# B&R Automation Studio project NAINV104C00R8L515F00 (part 9)

#### Act_Main_P0201.st
```iecst
(** 2018-12-21 **)
ACTION Act_Main_P0201:
	//LF width 2
	IF p_tyNtParamCurr.bLFProdWidth2Prep THEN
		fUIInRtStatOff(ADR(tyP0201OpsConv.tyOps.tyNumProdWidth2.uiRtStat));
		fUIInRtStatHide(ADR(tyP0201OpsConv.tyOps.tyNumProdWidth.uiRtStat));
	ELSE
		fUIInRtStatHide(ADR(tyP0201OpsConv.tyOps.tyNumProdWidth2.uiRtStat));
		fUIInRtStatOff(ADR(tyP0201OpsConv.tyOps.tyNumProdWidth.uiRtStat));
	END_IF

	IF p_tyNtParamCurr.tyDOSettings.diTLGreen<>0 OR p_tyNtParamCurr.tyDOSettings.diTLAmber<>0 OR p_tyNtParamCurr.tyDOSettings.diTLRed<>0 THEN
		IF p_tyNtParamCurr.eTLBuzMode=TLBuzModBHTC THEN
			tyP0201OpsConv.tyOps.tyBitmapMc.usiValueIdx := 200;
		ELSE
			tyP0201OpsConv.tyOps.tyBitmapMc.usiValueIdx := 100;
		END_IF
	ELSE
		tyP0201OpsConv.tyOps.tyBitmapMc.usiValueIdx := 0;
	END_IF

	fUIInRtStatHide(ADR(tyP0200OpsGen.tyOps.tyTxtLdrInActiveCtrl.uiRtStat));
	fUIInRtStatHide(ADR(tyP0201OpsConv.tyOps.tyTxtLdrInActiveCtrl.uiRtStat));
	fUIInRtStatHide(ADR(tyP0200OpsGen.tyOps.tyBitmapWarningLF.uiRtStat));
	fUIInRtStatHide(ADR(tyP0201OpsConv.tyOps.tyBitmapWarningLF.uiRtStat));

	//IO Monitor Standard
	//Digital Input Used
	IF p_tyNtParamCurr.tyDISettings.diSafetyRlySig = 0 THEN
		fUIInRtStatHide(ADR(tyP0201OpsConv.tyIOMonitor.tyBtnSafetyRlySig.uiRtStat));
	END_IF

	IF p_tyNtParamCurr.tyDISettings.diEStopSig = 0 THEN
		fUIInRtStatHide(ADR(tyP0201OpsConv.tyIOMonitor.tyBtnEStop.uiRtStat));
	END_IF

	IF p_tyNtParamCurr.tyDISettings.diCoverSWSig = 0 THEN
		fUIInRtStatHide(ADR(tyP0201OpsConv.tyIOMonitor.tyBtnCoverSWSig.uiRtStat));
	END_IF

	IF p_tyNtParamCurr.tyDISettings.diUBA = 0 THEN
		fUIInRtStatHide(ADR(tyP0201OpsConv.tyIOMonitor.tyBtnUBA.uiRtStat));
	END_IF

	IF p_tyNtParamCurr.tyDISettings.diDSB = 0 THEN
		fUIInRtStatHide(ADR(tyP0201OpsConv.tyIOMonitor.tyBtnDSB.uiRtStat));
	END_IF

	IF p_tyNtParamCurr.tyDISettings.diUBAStat = FALSE THEN
		fUIInRtStatHide(ADR(tyP0201OpsConv.tyIOMonitor.tyBtnUBAStat.uiRtStat));
	END_IF

	IF p_tyNtParamCurr.tyDISettings.diConvLftSen = 0 THEN
		fUIInRtStatHide(ADR(tyP0201OpsConv.tyIOMonitor.tyBtnConvLftSen.uiRtStat));
	END_IF

	IF p_tyNtParamCurr.tyDISettings.diConvRgtSen = 0 THEN
		fUIInRtStatHide(ADR(tyP0201OpsConv.tyIOMonitor.tyBtnConvRgtSen.uiRtStat));
	END_IF

	IF p_tyNtParamCurr.tyDISettings.diPressureSW = 0 THEN
		fUIInRtStatHide(ADR(tyP0201OpsConv.tyIOMonitor.tyBtnPressureSW.uiRtStat));
	END_IF

	IF p_tyNtParamCurr.tyDISettings.diThermalPrtSig = 0 THEN
		fUIInRtStatHide(ADR(tyP0201OpsConv.tyIOMonitor.tyBtnThermalPrtSig.uiRtStat));
	END_IF

	IF p_tyNtParamCurr.tyDISettings.diCoatingSen = 0 THEN
		fUIInRtStatHide(ADR(tyP0201OpsConv.tyIOMonitor.tyBtnCoatingSen.uiRtStat));
	END_IF

	IF p_tyNtParamCurr.tyDISettings.diUSWidthChkSen = 0 THEN
		fUIInRtStatHide(ADR(tyP0201OpsConv.tyIOMonitor.tyBtnUSWidthChkSen.uiRtStat));
	END_IF

	IF p_tyNtParamCurr.tyDISettings.diDSWidthChkSen = 0 THEN
		fUIInRtStatHide(ADR(tyP0201OpsConv.tyIOMonitor.tyBtnDSWidthChkSen.uiRtStat));
	END_IF

	IF p_tyNtParamCurr.tyDISettings.diInvertHomeSen = 0 THEN
		fUIInRtStatHide(ADR(tyP0201OpsConv.tyIOMonitor.tyBtnInvertHomeSen.uiRtStat));
	END_IF

	IF p_tyNtParamCurr.tyDISettings.diInvertRemoteSen = 0 THEN
		fUIInRtStatHide(ADR(tyP0201OpsConv.tyIOMonitor.tyBtnInvertRemoteSen.uiRtStat));
	END_IF

	IF p_tyNtParamCurr.tyDISettings.diInShutterOpenRS = 0 THEN
		fUIInRtStatHide(ADR(tyP0201OpsConv.tyIOMonitor.tyBtnInletShutterOpenRS.uiRtStat));
	END_IF

	IF p_tyNtParamCurr.tyDISettings.diInShutterCloseRS = 0 THEN
		fUIInRtStatHide(ADR(tyP0201OpsConv.tyIOMonitor.tyBtnInletShutterCloseRS.uiRtStat));
	END_IF

	IF p_tyNtParamCurr.tyDISettings.diOutShutterOpenRS = 0 THEN
		fUIInRtStatHide(ADR(tyP0201OpsConv.tyIOMonitor.tyBtnOutletShutterOpenRS.uiRtStat));
	END_IF

	IF p_tyNtParamCurr.tyDISettings.diOutShutterCloseRS = 0 THEN
		fUIInRtStatHide(ADR(tyP0201OpsConv.tyIOMonitor.tyBtnOutletShutterCloseRS.uiRtStat));
	END_IF

	//Digital Output Selected
	IF p_tyNtParamCurr.tyDOSettings.diSafetyRlyRst = 0 THEN
		fUIInRtStatHide(ADR(tyP0201OpsConv.tyIOMonitor.tyBtnSafetyRlyRst.uiRtStat));
	END_IF

	IF p_tyNtParamCurr.tyDOSettings.diTLGreen = 0 THEN
		fUIInRtStatHide(ADR(tyP0201OpsConv.tyIOMonitor.tyBtnTLGreen.uiRtStat));
	END_IF

	IF p_tyNtParamCurr.tyDOSettings.diTLAmber = 0 THEN
		fUIInRtStatHide(ADR(tyP0201OpsConv.tyIOMonitor.tyBtnTLAmber.uiRtStat));
	END_IF

	IF p_tyNtParamCurr.tyDOSettings.diTLRed = 0 THEN
		fUIInRtStatHide(ADR(tyP0201OpsConv.tyIOMonitor.tyBtnTLRed.uiRtStat));
	END_IF

	IF p_tyNtParamCurr.tyDOSettings.diTLWhite = 0 THEN
		fUIInRtStatHide(ADR(tyP0201OpsConv.tyIOMonitor.tyBtnTLWhite.uiRtStat));
	END_IF

	IF p_tyNtParamCurr.tyDOSettings.diTLBlue = 0 THEN
		fUIInRtStatHide(ADR(tyP0201OpsConv.tyIOMonitor.tyBtnTLBlue.uiRtStat));
	END_IF

	IF p_tyNtParamCurr.tyDOSettings.diBuz = 0 THEN
		fUIInRtStatHide(ADR(tyP0201OpsConv.tyIOMonitor.tyBtnBuzzer.uiRtStat));
	END_IF

	IF p_tyNtParamCurr.tyDOSettings.diCoatingStprRet = 0 THEN
		fUIInRtStatHide(ADR(tyP0201OpsConv.tyIOMonitor.tyBtnCoatingRetCtrl.uiRtStat));
	END_IF

	IF p_tyNtParamCurr.tyDOSettings.diUSB = 0 THEN
		fUIInRtStatHide(ADR(tyP0201OpsConv.tyIOMonitor.tyBtnUSB.uiRtStat));
	END_IF

	IF p_tyNtParamCurr.tyDOSettings.diDBA = 0 THEN
		fUIInRtStatHide(ADR(tyP0201OpsConv.tyIOMonitor.tyBtnDBA.uiRtStat));
	END_IF

	IF p_tyNtParamCurr.tyDOSettings.diDBAStat = 0 THEN
		fUIInRtStatHide(ADR(tyP0201OpsConv.tyIOMonitor.tyBtnDBAStat.uiRtStat));
	END_IF

	IF p_tyNtParamCurr.tyDOSettings.diConvMtrCW = 0 THEN
		fUIInRtStatHide(ADR(tyP0201OpsConv.tyIOMonitor.tyBtnConvMtrCW.uiRtStat));
	END_IF

	IF p_tyNtParamCurr.tyDOSettings.diConvMtrCCW = 0 THEN
		fUIInRtStatHide(ADR(tyP0201OpsConv.tyIOMonitor.tyBtnConvMtrCCW.uiRtStat));
	END_IF

	IF p_tyNtParamCurr.tyDOSettings.diStprUnblkCtrl = 0 THEN
		fUIInRtStatHide(ADR(tyP0201OpsConv.tyIOMonitor.tyBtnStprUnblkCtrl.uiRtStat));
	END_IF

	IF p_tyNtParamCurr.tyDOSettings.diStprBlkCtrl = 0 THEN
		fUIInRtStatHide(ADR(tyP0201OpsConv.tyIOMonitor.tyBtnStprBlkCtrl.uiRtStat));
	END_IF

	IF p_tyNtParamCurr.tyDOSettings.diInvertBrake = 0 THEN
		fUIInRtStatHide(ADR(tyP0201OpsConv.tyIOMonitor.tyBtnInvertBrake.uiRtStat));
	END_IF

	IF p_tyNtParamCurr.tyDOSettings.diInvertHome = 0 THEN
		fUIInRtStatHide(ADR(tyP0201OpsConv.tyIOMonitor.tyBtnInvertHome.uiRtStat));
	END_IF

	IF p_tyNtParamCurr.tyDOSettings.diInvertRemote = 0 THEN
		fUIInRtStatHide(ADR(tyP0201OpsConv.tyIOMonitor.tyBtnInvertRemote.uiRtStat));
	END_IF

	IF p_tyNtParamCurr.tyDOSettings.diMtrPwrRly = 0 THEN
		fUIInRtStatHide(ADR(tyP0201OpsConv.tyIOMonitor.tyBtnMtrPwrRly.uiRtStat));
	END_IF

	IF p_tyNtParamCurr.tyDOSettings.diClampControl = 0 THEN
		fUIInRtStatHide(ADR(tyP0201OpsConv.tyIOMonitor.tyBtnClampCtrl.uiRtStat));
	END_IF

	IF p_tyNtParamCurr.tyDOSettings.diUnclampControl = 0 THEN
		fUIInRtStatHide(ADR(tyP0201OpsConv.tyIOMonitor.tyBtnUnclampCtrl.uiRtStat));
	END_IF

	IF p_tyNtParamCurr.tyDOSettings.diInShutterOpenCtrl = 0 THEN
		fUIInRtStatHide(ADR(tyP0201OpsConv.tyIOMonitor.tyBtnInShutterOpenCtrl.uiRtStat));
	END_IF

	IF p_tyNtParamCurr.tyDOSettings.diInShutterCloseCtrl = 0 THEN
		fUIInRtStatHide(ADR(tyP0201OpsConv.tyIOMonitor.tyBtnInShutterCloseCtrl.uiRtStat));
	END_IF

	IF p_tyNtParamCurr.tyDOSettings.diOutShutterOpenCtrl = 0 THEN
		fUIInRtStatHide(ADR(tyP0201OpsConv.tyIOMonitor.tyBtnOutShutterOpenCtrl.uiRtStat));
	END_IF

	IF p_tyNtParamCurr.tyDOSettings.diOutShutterCloseCtrl = 0 THEN
		fUIInRtStatHide(ADR(tyP0201OpsConv.tyIOMonitor.tyBtnOutShutterCloseCtrl.uiRtStat));
	END_IF

	//IO Monitor Non Standard
	//Digital Input Used
	IF p_tyNtParamCurr.tyDISettings.diSafetyRlySig = 0 THEN
		fUIInRtStatHide(ADR(tyP0201OpsConv.tyIOMonitorXStd.tyBtnSafetyRlySig.uiRtStat));
	END_IF

	IF p_tyNtParamCurr.tyDISettings.diEStopSig = 0 THEN
		fUIInRtStatHide(ADR(tyP0201OpsConv.tyIOMonitorXStd.tyBtnEStop.uiRtStat));
	END_IF

	IF p_tyNtParamCurr.tyDISettings.diCoverSWSig = 0 THEN
		fUIInRtStatHide(ADR(tyP0201OpsConv.tyIOMonitorXStd.tyBtnCoverSWSig.uiRtStat));
	END_IF

	IF p_tyNtParamCurr.tyDISettings.diUBA = 0 THEN
		fUIInRtStatHide(ADR(tyP0201OpsConv.tyIOMonitorXStd.tyBtnUBA.uiRtStat));
	END_IF

	IF p_tyNtParamCurr.tyDISettings.diUBA2 = 0 THEN
		fUIInRtStatHide(ADR(tyP0201OpsConv.tyIOMonitorXStd.tyBtnUBA2.uiRtStat));
	END_IF

	IF p_tyNtParamCurr.tyDISettings.diDSB = 0 THEN
		fUIInRtStatHide(ADR(tyP0201OpsConv.tyIOMonitorXStd.tyBtnDSB.uiRtStat));
	END_IF

	IF p_tyNtParamCurr.tyDISettings.diUBAStat = FALSE THEN
		fUIInRtStatHide(ADR(tyP0201OpsConv.tyIOMonitorXStd.tyBtnUBAStat.uiRtStat));
	END_IF

	IF p_tyNtParamCurr.tyDISettings.diUBAStat2 = FALSE THEN
		fUIInRtStatHide(ADR(tyP0201OpsConv.tyIOMonitorXStd.tyBtnUBAStat2.uiRtStat));
	END_IF

	IF p_tyNtParamCurr.tyDISettings.diConvLftSen = 0 THEN
		fUIInRtStatHide(ADR(tyP0201OpsConv.tyIOMonitorXStd.tyBtnConvLftSen.uiRtStat));
	END_IF

	IF p_tyNtParamCurr.tyDISettings.diConvRgtSen = 0 THEN
		fUIInRtStatHide(ADR(tyP0201OpsConv.tyIOMonitorXStd.tyBtnConvRgtSen.uiRtStat));
	END_IF

	IF p_tyNtParamCurr.tyDISettings.diPressureSW = 0 THEN
		fUIInRtStatHide(ADR(tyP0201OpsConv.tyIOMonitorXStd.tyBtnPressureSW.uiRtStat));
	END_IF

	IF p_tyNtParamCurr.tyDISettings.diThermalPrtSig = 0 THEN
		fUIInRtStatHide(ADR(tyP0201OpsConv.tyIOMonitorXStd.tyBtnThermalPrtSig.uiRtStat));
	END_IF

	IF p_tyNtParamCurr.tyDISettings.diCoatingSen = 0 THEN
		fUIInRtStatHide(ADR(tyP0201OpsConv.tyIOMonitorXStd.tyBtnCoatingSen.uiRtStat));
	END_IF

	IF p_tyNtParamCurr.tyDISettings.diUSWidthChkSen = 0 THEN
		fUIInRtStatHide(ADR(tyP0201OpsConv.tyIOMonitorXStd.tyBtnUSWidthChkSen.uiRtStat));
	END_IF

	IF p_tyNtParamCurr.tyDISettings.diDSWidthChkSen = 0 THEN
		fUIInRtStatHide(ADR(tyP0201OpsConv.tyIOMonitorXStd.tyBtnDSWidthChkSen.uiRtStat));
	END_IF

	IF p_tyNtParamCurr.tyDISettings.diInvertHomeSen = 0 THEN
		fUIInRtStatHide(ADR(tyP0201OpsConv.tyIOMonitorXStd.tyBtnInvertHomeSen.uiRtStat));
	END_IF

	IF p_tyNtParamCurr.tyDISettings.diInvertRemoteSen = 0 THEN
		fUIInRtStatHide(ADR(tyP0201OpsConv.tyIOMonitorXStd.tyBtnInvertRemoteSen.uiRtStat));
	END_IF

	IF p_tyNtParamCurr.tyDISettings.diInShutterOpenRS = 0 THEN
		fUIInRtStatHide(ADR(tyP0201OpsConv.tyIOMonitorXStd.tyBtnInletShutterOpenRS.uiRtStat));
	END_IF

	IF p_tyNtParamCurr.tyDISettings.diInShutterCloseRS = 0 THEN
		fUIInRtStatHide(ADR(tyP0201OpsConv.tyIOMonitorXStd.tyBtnInletShutterCloseRS.uiRtStat));
	END_IF

	IF p_tyNtParamCurr.tyDISettings.diOutShutterOpenRS = 0 THEN
		fUIInRtStatHide(ADR(tyP0201OpsConv.tyIOMonitorXStd.tyBtnOutletShutterOpenRS.uiRtStat));
	END_IF

	IF p_tyNtParamCurr.tyDISettings.diOutShutterCloseRS = 0 THEN
		fUIInRtStatHide(ADR(tyP0201OpsConv.tyIOMonitorXStd.tyBtnOutletShutterCloseRS.uiRtStat));
	END_IF

	IF p_tyNtParamCurr.tyDISettings.diClamp2Sen = 0 THEN
		fUIInRtStatHide(ADR(tyP0201OpsConv.tyIOMonitorXStd.tyBtnClamp2Sen.uiRtStat));
	END_IF

	IF p_tyNtParamCurr.tyDISettings.diClamp3Sen = 0 THEN
		fUIInRtStatHide(ADR(tyP0201OpsConv.tyIOMonitorXStd.tyBtnClamp3Sen.uiRtStat));
	END_IF

	IF p_tyNtParamCurr.tyDISettings.diClampRS1 = 0 THEN
		fUIInRtStatHide(ADR(tyP0201OpsConv.tyIOMonitorXStd.tyBtnClampRS1.uiRtStat));
	END_IF

	IF p_tyNtParamCurr.tyDISettings.diUnClampRS1 = 0 THEN
		fUIInRtStatHide(ADR(tyP0201OpsConv.tyIOMonitorXStd.tyBtnUnClampRS1.uiRtStat));
	END_IF

	IF p_tyNtParamCurr.tyDISettings.diClampRS2 = 0 THEN
		fUIInRtStatHide(ADR(tyP0201OpsConv.tyIOMonitorXStd.tyBtnClampRS2.uiRtStat));
	END_IF

	IF p_tyNtParamCurr.tyDISettings.diUnClampRS2 = 0 THEN
		fUIInRtStatHide(ADR(tyP0201OpsConv.tyIOMonitorXStd.tyBtnUnClampRS2.uiRtStat));
	END_IF

	IF p_tyNtParamCurr.tyDISettings.diClampRS3 = 0 THEN
		fUIInRtStatHide(ADR(tyP0201OpsConv.tyIOMonitorXStd.tyBtnClampRS3.uiRtStat));
	END_IF

	IF p_tyNtParamCurr.tyDISettings.diUnClampRS3 = 0 THEN
		fUIInRtStatHide(ADR(tyP0201OpsConv.tyIOMonitorXStd.tyBtnUnClampRS3.uiRtStat));
	END_IF

	//Digital Output Selected
	IF p_tyNtParamCurr.tyDOSettings.diSafetyRlyRst = 0 THEN
		fUIInRtStatHide(ADR(tyP0201OpsConv.tyIOMonitorXStd.tyBtnSafetyRlyRst.uiRtStat));
	END_IF

	IF p_tyNtParamCurr.tyDOSettings.diTLGreen = 0 THEN
		fUIInRtStatHide(ADR(tyP0201OpsConv.tyIOMonitorXStd.tyBtnTLGreen.uiRtStat));
	END_IF

	IF p_tyNtParamCurr.tyDOSettings.diTLAmber = 0 THEN
		fUIInRtStatHide(ADR(tyP0201OpsConv.tyIOMonitorXStd.tyBtnTLAmber.uiRtStat));
	END_IF

	IF p_tyNtParamCurr.tyDOSettings.diTLRed = 0 THEN
		fUIInRtStatHide(ADR(tyP0201OpsConv.tyIOMonitorXStd.tyBtnTLRed.uiRtStat));
	END_IF

	IF p_tyNtParamCurr.tyDOSettings.diTLWhite = 0 THEN
		fUIInRtStatHide(ADR(tyP0201OpsConv.tyIOMonitorXStd.tyBtnTLWhite.uiRtStat));
	END_IF

	IF p_tyNtParamCurr.tyDOSettings.diTLBlue = 0 THEN
		fUIInRtStatHide(ADR(tyP0201OpsConv.tyIOMonitorXStd.tyBtnTLBlue.uiRtStat));
	END_IF

	IF p_tyNtParamCurr.tyDOSettings.diBuz = 0 THEN
		fUIInRtStatHide(ADR(tyP0201OpsConv.tyIOMonitorXStd.tyBtnBuzzer.uiRtStat));
	END_IF

	IF p_tyNtParamCurr.tyDOSettings.diCoatingStprRet = 0 THEN
		fUIInRtStatHide(ADR(tyP0201OpsConv.tyIOMonitorXStd.tyBtnCoatingRetCtrl.uiRtStat));
	END_IF

	IF p_tyNtParamCurr.tyDOSettings.diUSB = 0 THEN
		fUIInRtStatHide(ADR(tyP0201OpsConv.tyIOMonitorXStd.tyBtnUSB.uiRtStat));
	END_IF

	IF p_tyNtParamCurr.tyDOSettings.diUSB2 = 0 THEN
		fUIInRtStatHide(ADR(tyP0201OpsConv.tyIOMonitorXStd.tyBtnUSB2.uiRtStat));
	END_IF

	IF p_tyNtParamCurr.tyDOSettings.diDBA = 0 THEN
		fUIInRtStatHide(ADR(tyP0201OpsConv.tyIOMonitorXStd.tyBtnDBA.uiRtStat));
	END_IF

	IF p_tyNtParamCurr.tyDOSettings.diDBAStat = 0 THEN
		fUIInRtStatHide(ADR(tyP0201OpsConv.tyIOMonitorXStd.tyBtnDBAStat.uiRtStat));
	END_IF

	IF p_tyNtParamCurr.tyDOSettings.diConvMtrCW = 0 THEN
		fUIInRtStatHide(ADR(tyP0201OpsConv.tyIOMonitorXStd.tyBtnConvMtrCW.uiRtStat));
	END_IF

	IF p_tyNtParamCurr.tyDOSettings.diConvMtrCCW = 0 THEN
		fUIInRtStatHide(ADR(tyP0201OpsConv.tyIOMonitorXStd.tyBtnConvMtrCCW.uiRtStat));
	END_IF

	IF p_tyNtParamCurr.tyDOSettings.diInvertBrake = 0 THEN
		fUIInRtStatHide(ADR(tyP0201OpsConv.tyIOMonitorXStd.tyBtnInvertBrake.uiRtStat));
	END_IF

	IF p_tyNtParamCurr.tyDOSettings.diInvertHome = 0 THEN
		fUIInRtStatHide(ADR(tyP0201OpsConv.tyIOMonitorXStd.tyBtnInvertHome.uiRtStat));
	END_IF

	IF p_tyNtParamCurr.tyDOSettings.diInvertRemote = 0 THEN
		fUIInRtStatHide(ADR(tyP0201OpsConv.tyIOMonitorXStd.tyBtnInvertRemote.uiRtStat));
	END_IF

	IF p_tyNtParamCurr.tyDOSettings.diMtrPwrRly = 0 THEN
		fUIInRtStatHide(ADR(tyP0201OpsConv.tyIOMonitorXStd.tyBtnMtrPwrRly.uiRtStat));
	END_IF

	IF p_tyNtParamCurr.tyDOSettings.diInShutterOpenCtrl = 0 THEN
		fUIInRtStatHide(ADR(tyP0201OpsConv.tyIOMonitorXStd.tyBtnInShutterOpenCtrl.uiRtStat));
	END_IF

	IF p_tyNtParamCurr.tyDOSettings.diInShutterCloseCtrl = 0 THEN
		fUIInRtStatHide(ADR(tyP0201OpsConv.tyIOMonitorXStd.tyBtnInShutterCloseCtrl.uiRtStat));
	END_IF

	IF p_tyNtParamCurr.tyDOSettings.diOutShutterOpenCtrl = 0 THEN
		fUIInRtStatHide(ADR(tyP0201OpsConv.tyIOMonitorXStd.tyBtnOutShutterOpenCtrl.uiRtStat));
	END_IF

	IF p_tyNtParamCurr.tyDOSettings.diOutShutterCloseCtrl = 0 THEN
		fUIInRtStatHide(ADR(tyP0201OpsConv.tyIOMonitorXStd.tyBtnOutShutterCloseCtrl.uiRtStat));
	END_IF

	IF p_tyNtParamCurr.tyDOSettings.diClamp1Ctrl = 0 THEN
		fUIInRtStatHide(ADR(tyP0201OpsConv.tyIOMonitorXStd.tyBtnClamp1Ctrl.uiRtStat));
	END_IF

	IF p_tyNtParamCurr.tyDOSettings.diUnClamp1Ctrl = 0 THEN
		fUIInRtStatHide(ADR(tyP0201OpsConv.tyIOMonitorXStd.tyBtnUnclamp1Ctrl.uiRtStat));
	END_IF

	IF p_tyNtParamCurr.tyDOSettings.diClamp2Ctrl = 0 THEN
		fUIInRtStatHide(ADR(tyP0201OpsConv.tyIOMonitorXStd.tyBtnClamp2Ctrl.uiRtStat));
	END_IF

	IF p_tyNtParamCurr.tyDOSettings.diUnClamp2Ctrl = 0 THEN
		fUIInRtStatHide(ADR(tyP0201OpsConv.tyIOMonitorXStd.tyBtnUnclamp2Ctrl.uiRtStat));
	END_IF

	IF p_tyNtParamCurr.tyDOSettings.diClamp3Ctrl = 0 THEN
		fUIInRtStatHide(ADR(tyP0201OpsConv.tyIOMonitorXStd.tyBtnClamp3Ctrl.uiRtStat));
	END_IF

	IF p_tyNtParamCurr.tyDOSettings.diUnClamp3Ctrl = 0 THEN
		fUIInRtStatHide(ADR(tyP0201OpsConv.tyIOMonitorXStd.tyBtnUnclamp3Ctrl.uiRtStat));
	END_IF

	//XStd Machine Safety
	//Digital Input Used
	IF p_tyNtParamCurr.tyDISettings.diSafetyRlySig = 0 THEN
		fUIInRtStatHide(ADR(tyP0201OpsConv.tyIOMonitorXStdMachineSafety.tyBtnSafetyRlySig.uiRtStat));
	END_IF

	IF p_tyNtParamCurr.tyDISettings.diEStopSig = 0 THEN
		fUIInRtStatHide(ADR(tyP0201OpsConv.tyIOMonitorXStdMachineSafety.tyBtnEStop.uiRtStat));
	END_IF

	IF p_tyNtParamCurr.tyDISettings.diCoverSWSig = 0 THEN
		fUIInRtStatHide(ADR(tyP0201OpsConv.tyIOMonitorXStdMachineSafety.tyBtnCoverSWSig.uiRtStat));
	END_IF

	IF p_tyNtParamCurr.tyDISettings.diUBA = 0 THEN
		fUIInRtStatHide(ADR(tyP0201OpsConv.tyIOMonitorXStdMachineSafety.tyBtnUBA.uiRtStat));
	END_IF

	IF p_tyNtParamCurr.tyDISettings.diDSB = 0 THEN
		fUIInRtStatHide(ADR(tyP0201OpsConv.tyIOMonitorXStdMachineSafety.tyBtnDSB.uiRtStat));
	END_IF

	IF p_tyNtParamCurr.tyDISettings.diUBAStat = FALSE THEN
		fUIInRtStatHide(ADR(tyP0201OpsConv.tyIOMonitorXStdMachineSafety.tyBtnUBAStat.uiRtStat));
	END_IF

	IF p_tyNtParamCurr.tyDISettings.diConvLftSen = 0 THEN
		fUIInRtStatHide(ADR(tyP0201OpsConv.tyIOMonitorXStdMachineSafety.tyBtnConvLftSen.uiRtStat));
	END_IF

	IF p_tyNtParamCurr.tyDISettings.diConvRgtSen = 0 THEN
		fUIInRtStatHide(ADR(tyP0201OpsConv.tyIOMonitorXStdMachineSafety.tyBtnConvRgtSen.uiRtStat));
	END_IF

	IF p_tyNtParamCurr.tyDISettings.diPressureSW = 0 THEN
		fUIInRtStatHide(ADR(tyP0201OpsConv.tyIOMonitorXStdMachineSafety.tyBtnPressureSW.uiRtStat));
	END_IF

	IF p_tyNtParamCurr.tyDISettings.diThermalPrtSig = 0 THEN
		fUIInRtStatHide(ADR(tyP0201OpsConv.tyIOMonitorXStdMachineSafety.tyBtnThermalPrtSig.uiRtStat));
	END_IF

	IF p_tyNtParamCurr.tyDISettings.diCoatingSen = 0 THEN
		fUIInRtStatHide(ADR(tyP0201OpsConv.tyIOMonitorXStdMachineSafety.tyBtnCoatingSen.uiRtStat));
	END_IF

	IF p_tyNtParamCurr.tyDISettings.diUSWidthChkSen = 0 THEN
		fUIInRtStatHide(ADR(tyP0201OpsConv.tyIOMonitorXStdMachineSafety.tyBtnUSWidthChkSen.uiRtStat));
	END_IF

	IF p_tyNtParamCurr.tyDISettings.diDSWidthChkSen = 0 THEN
		fUIInRtStatHide(ADR(tyP0201OpsConv.tyIOMonitorXStdMachineSafety.tyBtnDSWidthChkSen.uiRtStat));
	END_IF

	IF p_tyNtParamCurr.tyDISettings.diInvertHomeSen = 0 THEN
		fUIInRtStatHide(ADR(tyP0201OpsConv.tyIOMonitorXStdMachineSafety.tyBtnInvertHomeSen.uiRtStat));
	END_IF

	IF p_tyNtParamCurr.tyDISettings.diInvertRemoteSen = 0 THEN
		fUIInRtStatHide(ADR(tyP0201OpsConv.tyIOMonitorXStdMachineSafety.tyBtnInvertRemoteSen.uiRtStat));
	END_IF

	IF p_tyNtParamCurr.tyDISettings.diInShutterOpenRS = 0 THEN
		fUIInRtStatHide(ADR(tyP0201OpsConv.tyIOMonitorXStdMachineSafety.tyBtnInletShutterOpenRS.uiRtStat));
	END_IF

	IF p_tyNtParamCurr.tyDISettings.diInShutterCloseRS = 0 THEN
		fUIInRtStatHide(ADR(tyP0201OpsConv.tyIOMonitorXStdMachineSafety.tyBtnInletShutterCloseRS.uiRtStat));
	END_IF

	IF p_tyNtParamCurr.tyDISettings.diOutShutterOpenRS = 0 THEN
		fUIInRtStatHide(ADR(tyP0201OpsConv.tyIOMonitorXStdMachineSafety.tyBtnOutletShutterOpenRS.uiRtStat));
	END_IF

	IF p_tyNtParamCurr.tyDISettings.diOutShutterCloseRS = 0 THEN
		fUIInRtStatHide(ADR(tyP0201OpsConv.tyIOMonitorXStdMachineSafety.tyBtnOutletShutterCloseRS.uiRtStat));
	END_IF

	IF p_tyNtParamCurr.tyDISettings.diClamp2Sen = 0 THEN
		fUIInRtStatHide(ADR(tyP0201OpsConv.tyIOMonitorXStdMachineSafety.tyBtnClamp2Sen.uiRtStat));
	END_IF

	IF p_tyNtParamCurr.tyDISettings.diClamp3Sen = 0 THEN
		fUIInRtStatHide(ADR(tyP0201OpsConv.tyIOMonitorXStdMachineSafety.tyBtnClamp3Sen.uiRtStat));
	END_IF

	IF p_tyNtParamCurr.tyDISettings.diClampRS1 = 0 THEN
		fUIInRtStatHide(ADR(tyP0201OpsConv.tyIOMonitorXStdMachineSafety.tyBtnClampRS1.uiRtStat));
	END_IF

	IF p_tyNtParamCurr.tyDISettings.diUnClampRS1 = 0 THEN
		fUIInRtStatHide(ADR(tyP0201OpsConv.tyIOMonitorXStdMachineSafety.tyBtnUnClampRS1.uiRtStat));
	END_IF

	IF p_tyNtParamCurr.tyDISettings.diClampRS2 = 0 THEN
		fUIInRtStatHide(ADR(tyP0201OpsConv.tyIOMonitorXStdMachineSafety.tyBtnClampRS2.uiRtStat));
	END_IF

	IF p_tyNtParamCurr.tyDISettings.diUnClampRS2 = 0 THEN
		fUIInRtStatHide(ADR(tyP0201OpsConv.tyIOMonitorXStdMachineSafety.tyBtnUnClampRS2.uiRtStat));
	END_IF

	IF p_tyNtParamCurr.tyDISettings.diClampRS3 = 0 THEN
		fUIInRtStatHide(ADR(tyP0201OpsConv.tyIOMonitorXStdMachineSafety.tyBtnClampRS3.uiRtStat));
	END_IF

	IF p_tyNtParamCurr.tyDISettings.diUnClampRS3 = 0 THEN
		fUIInRtStatHide(ADR(tyP0201OpsConv.tyIOMonitorXStdMachineSafety.tyBtnUnClampRS3.uiRtStat));
	END_IF
	// ADD
	IF p_tyNtParamCurr.tyDISettings.diCoverSWSig2 = 0 THEN
		fUIInRtStatHide(ADR(tyP0201OpsConv.tyIOMonitorXStdMachineSafety.tyBtnCoverSWSig2.uiRtStat));
	END_IF

	IF p_tyNtParamCurr.tyDISettings.diSafetySigFromUS = 0 THEN
		fUIInRtStatHide(ADR(tyP0201OpsConv.tyIOMonitorXStdMachineSafety.tyBtnSafetySigFromUS.uiRtStat));
	END_IF

	IF p_tyNtParamCurr.tyDISettings.diSafetySigFromDS = 0 THEN
		fUIInRtStatHide(ADR(tyP0201OpsConv.tyIOMonitorXStdMachineSafety.tyBtnSafetySigFromDS.uiRtStat));
	END_IF

	IF p_tyNtParamCurr.tyDISettings.diUnlockCoverSigFromUS = 0 THEN
		fUIInRtStatHide(ADR(tyP0201OpsConv.tyIOMonitorXStdMachineSafety.tyBtnUnlockCoverSigFromUS.uiRtStat));
	END_IF

	IF p_tyNtParamCurr.tyDISettings.diUnlockCoverSigFromDS = 0 THEN
		fUIInRtStatHide(ADR(tyP0201OpsConv.tyIOMonitorXStdMachineSafety.tyBtnUnlockCoverSigFromDS.uiRtStat));
	END_IF

	IF p_tyNtParamCurr.tyDISettings.diCoverUnlockPB1 = 0 THEN
		fUIInRtStatHide(ADR(tyP0201OpsConv.tyIOMonitorXStdMachineSafety.tyBtnCoverUnlockPB1.uiRtStat));
	END_IF

	//Digital Output Selected
	IF p_tyNtParamCurr.tyDOSettings.diSafetyRlyRst = 0 THEN
		fUIInRtStatHide(ADR(tyP0201OpsConv.tyIOMonitorXStdMachineSafety.tyBtnSafetyRlyRst.uiRtStat));
	END_IF

	IF p_tyNtParamCurr.tyDOSettings.diTLGreen = 0 THEN
		fUIInRtStatHide(ADR(tyP0201OpsConv.tyIOMonitorXStdMachineSafety.tyBtnTLGreen.uiRtStat));
	END_IF

	IF p_tyNtParamCurr.tyDOSettings.diTLAmber = 0 THEN
		fUIInRtStatHide(ADR(tyP0201OpsConv.tyIOMonitorXStdMachineSafety.tyBtnTLAmber.uiRtStat));
	END_IF

	IF p_tyNtParamCurr.tyDOSettings.diTLRed = 0 THEN
		fUIInRtStatHide(ADR(tyP0201OpsConv.tyIOMonitorXStdMachineSafety.tyBtnTLRed.uiRtStat));
	END_IF

	IF p_tyNtParamCurr.tyDOSettings.diTLWhite = 0 THEN
		fUIInRtStatHide(ADR(tyP0201OpsConv.tyIOMonitorXStdMachineSafety.tyBtnTLWhite.uiRtStat));
	END_IF

	IF p_tyNtParamCurr.tyDOSettings.diTLBlue = 0 THEN
		fUIInRtStatHide(ADR(tyP0201OpsConv.tyIOMonitorXStdMachineSafety.tyBtnTLBlue.uiRtStat));
	END_IF

	IF p_tyNtParamCurr.tyDOSettings.diBuz = 0 THEN
		fUIInRtStatHide(ADR(tyP0201OpsConv.tyIOMonitorXStdMachineSafety.tyBtnBuzzer.uiRtStat));
	END_IF

	IF p_tyNtParamCurr.tyDOSettings.diCoatingStprRet = 0 THEN
		fUIInRtStatHide(ADR(tyP0201OpsConv.tyIOMonitorXStdMachineSafety.tyBtnCoatingRetCtrl.uiRtStat));
	END_IF

	IF p_tyNtParamCurr.tyDOSettings.diUSB = 0 THEN
		fUIInRtStatHide(ADR(tyP0201OpsConv.tyIOMonitorXStdMachineSafety.tyBtnUSB.uiRtStat));
	END_IF

	IF p_tyNtParamCurr.tyDOSettings.diDBA = 0 THEN
		fUIInRtStatHide(ADR(tyP0201OpsConv.tyIOMonitorXStdMachineSafety.tyBtnDBA.uiRtStat));
	END_IF

	IF p_tyNtParamCurr.tyDOSettings.diDBAStat = 0 THEN
		fUIInRtStatHide(ADR(tyP0201OpsConv.tyIOMonitorXStdMachineSafety.tyBtnDBAStat.uiRtStat));
	END_IF

	IF p_tyNtParamCurr.tyDOSettings.diConvMtrCW = 0 THEN
		fUIInRtStatHide(ADR(tyP0201OpsConv.tyIOMonitorXStdMachineSafety.tyBtnConvMtrCW.uiRtStat));
	END_IF

	IF p_tyNtParamCurr.tyDOSettings.diConvMtrCCW = 0 THEN
		fUIInRtStatHide(ADR(tyP0201OpsConv.tyIOMonitorXStdMachineSafety.tyBtnConvMtrCCW.uiRtStat));
	END_IF

	IF p_tyNtParamCurr.tyDOSettings.diInvertBrake = 0 THEN
		fUIInRtStatHide(ADR(tyP0201OpsConv.tyIOMonitorXStdMachineSafety.tyBtnInvertBrake.uiRtStat));
	END_IF

	IF p_tyNtParamCurr.tyDOSettings.diInvertHome = 0 THEN
		fUIInRtStatHide(ADR(tyP0201OpsConv.tyIOMonitorXStdMachineSafety.tyBtnInvertHome.uiRtStat));
	END_IF

	IF p_tyNtParamCurr.tyDOSettings.diInvertRemote = 0 THEN
		fUIInRtStatHide(ADR(tyP0201OpsConv.tyIOMonitorXStdMachineSafety.tyBtnInvertRemote.uiRtStat));
	END_IF

	IF p_tyNtParamCurr.tyDOSettings.diMtrPwrRly = 0 THEN
		fUIInRtStatHide(ADR(tyP0201OpsConv.tyIOMonitorXStdMachineSafety.tyBtnMtrPwrRly.uiRtStat));
	END_IF

	IF p_tyNtParamCurr.tyDOSettings.diInShutterOpenCtrl = 0 THEN
		fUIInRtStatHide(ADR(tyP0201OpsConv.tyIOMonitorXStdMachineSafety.tyBtnInShutterOpenCtrl.uiRtStat));
	END_IF

	IF p_tyNtParamCurr.tyDOSettings.diInShutterCloseCtrl = 0 THEN
		fUIInRtStatHide(ADR(tyP0201OpsConv.tyIOMonitorXStdMachineSafety.tyBtnInShutterCloseCtrl.uiRtStat));
	END_IF

	IF p_tyNtParamCurr.tyDOSettings.diOutShutterOpenCtrl = 0 THEN
		fUIInRtStatHide(ADR(tyP0201OpsConv.tyIOMonitorXStdMachineSafety.tyBtnOutShutterOpenCtrl.uiRtStat));
	END_IF

	IF p_tyNtParamCurr.tyDOSettings.diOutShutterCloseCtrl = 0 THEN
		fUIInRtStatHide(ADR(tyP0201OpsConv.tyIOMonitorXStdMachineSafety.tyBtnOutShutterCloseCtrl.uiRtStat));
	END_IF

	IF p_tyNtParamCurr.tyDOSettings.diClamp1Ctrl = 0 THEN
		fUIInRtStatHide(ADR(tyP0201OpsConv.tyIOMonitorXStdMachineSafety.tyBtnClamp1Ctrl.uiRtStat));
	END_IF

	IF p_tyNtParamCurr.tyDOSettings.diUnClamp1Ctrl = 0 THEN
		fUIInRtStatHide(ADR(tyP0201OpsConv.tyIOMonitorXStdMachineSafety.tyBtnUnclamp1Ctrl.uiRtStat));
	END_IF

	IF p_tyNtParamCurr.tyDOSettings.diClamp2Ctrl = 0 THEN
		fUIInRtStatHide(ADR(tyP0201OpsConv.tyIOMonitorXStdMachineSafety.tyBtnClamp2Ctrl.uiRtStat));
	END_IF

	IF p_tyNtParamCurr.tyDOSettings.diUnClamp2Ctrl = 0 THEN
		fUIInRtStatHide(ADR(tyP0201OpsConv.tyIOMonitorXStdMachineSafety.tyBtnUnclamp2Ctrl.uiRtStat));
	END_IF

	IF p_tyNtParamCurr.tyDOSettings.diClamp3Ctrl = 0 THEN
		fUIInRtStatHide(ADR(tyP0201OpsConv.tyIOMonitorXStdMachineSafety.tyBtnClamp3Ctrl.uiRtStat));
	END_IF

	IF p_tyNtParamCurr.tyDOSettings.diUnClamp3Ctrl = 0 THEN
		fUIInRtStatHide(ADR(tyP0201OpsConv.tyIOMonitorXStdMachineSafety.tyBtnUnclamp3Ctrl.uiRtStat));
	END_IF

	// ADD
	IF p_tyNtParamCurr.tyDOSettings.diTopCvrUnlckToDS = 0 THEN
		fUIInRtStatHide(ADR(tyP0201OpsConv.tyIOMonitorXStdMachineSafety.tyBtnTopCvrUnlckToDS.uiRtStat));
	END_IF

	IF p_tyNtParamCurr.tyDOSettings.diTopCvrUnlckToUS = 0 THEN    //diTopCvrUnlckToUS
		fUIInRtStatHide(ADR(tyP0201OpsConv.tyIOMonitorXStdMachineSafety.tyBtnTopCvrUnlckToUS.uiRtStat)); // follow DS (single output)
	END_IF

	IF p_tyNtParamCurr.tyDOSettings.diMachineSafetySigToDS = 0 THEN
		fUIInRtStatHide(ADR(tyP0201OpsConv.tyIOMonitorXStdMachineSafety.tyBtniMachineSafetySigToDS.uiRtStat));
	END_IF

	IF p_tyNtParamCurr.tyDOSettings.diMachineSafetySigToUS = 0 THEN
		fUIInRtStatHide(ADR(tyP0201OpsConv.tyIOMonitorXStdMachineSafety.tyBtnMachineSafetySigToUS.uiRtStat));
	END_IF

	IF p_tyNtParamCurr.tyDOSettings.diCoverPBLED1 = 0 THEN
		fUIInRtStatHide(ADR(tyP0201OpsConv.tyIOMonitorXStdMachineSafety.tyBtnPBLED1.uiRtStat));
	END_IF

	IF p_tyNtParamCurr.tyDOSettings.diBypassTopCover1 = 0 THEN
		fUIInRtStatHide(ADR(tyP0201OpsConv.tyIOMonitorXStdMachineSafety.tyBtnBypassTopCover1.uiRtStat));
	END_IF

	IF p_tyNtParamCurr.tyDOSettings.diSafetyTopCoverSWCoil1 = 0 THEN
		fUIInRtStatHide(ADR(tyP0201OpsConv.tyIOMonitorXStdMachineSafety.tyBtnSafetyTopCoverSWCoil1.uiRtStat));
	END_IF

	//Change Parameter
	tyP0201OpsConv.tyChgParam.tyDrpDnMcMode.usiValueMinIdx	:= DINT_TO_USINT(p_tyNtParamCurr.tyProdRcpMcModLmt.diMin);
	tyP0201OpsConv.tyChgParam.tyDrpDnMcMode.usiValueMaxIdx	:= DINT_TO_USINT(p_tyNtParamCurr.tyProdRcpMcModLmt.diMax);

	tyP0201OpsConv.tyChgParam.tyNumProdWidth.diValueMin		:= p_tyNtParamCurr.tyProdRcpWidthLmt.diMin;
	tyP0201OpsConv.tyChgParam.tyNumProdWidth.diValueMax		:= p_tyNtParamCurr.tyProdRcpWidthLmt.diMax;

	tyP0201OpsConv.tyChgParam.tyDrpDnFlippedBrd.usiValueMinIdx	:= DINT_TO_USINT(p_tyNtParamCurr.tyProdRcpFlippedBrdLmt.diMin);
	tyP0201OpsConv.tyChgParam.tyDrpDnFlippedBrd.usiValueMaxIdx	:= DINT_TO_USINT(p_tyNtParamCurr.tyProdRcpFlippedBrdLmt.diMax);

	//Display

	tyP0201OpsConv.tyChgParam.tyDrpDnFlippedBrd.uiRtStat.0 := NOT p_tyNtParamCurr.bHermesPrep;

	tyP0201OpsConv.tyOps.tyLblFlippedBrd.uiRtStat.0 := NOT p_tyNtParamCurr.bHermesPrep;
	tyP0201OpsConv.tyOps.tyTxtFlippedBrd.uiRtStat.0 := NOT p_tyNtParamCurr.bHermesPrep;
	tyP0201OpsConv.tyOps.tyBtnBypassTopCover1.uiRtStat.0 := NOT(p_tyNtParamCurr.bUnlockCoverPrep);
END_ACTION
```

#### Act_Main_P0300.st
```iecst
(** 2018-12-21 **)
ACTION Act_Main_P0300:

	//Display
	tyP0300McInfo.tyMcInfo.tyStringSoftwareVer.sValue	:= sSWVersion;
	tyP0300McInfo.tyMcInfo.tyTxtNtAddr.usiValueIdx		:= p_tyNtParamCurr.usiNtAddr;
	tyP0300McInfo.tyMcInfo.tyStringJobNo.sValue			:= CONCAT('(', CONCAT(p_tyNtParamCurr.sJobNo, ')'));

END_ACTION
```

#### Act_Main_P0400.st
```iecst
(** 2018-12-21 **)
ACTION Act_Main_P0400:
	//Display
//	tyP0400ProdSel.tyProdSel.tyTxtFlippedBrd.uiRtStat.0	:= NOT p_tyNtParamCurr.bHermesPrep;
//	tyP0400ProdSel.tyRcpDet.tyTxtFlippedBrd.uiRtStat.0	:= NOT p_tyNtParamCurr.bHermesPrep;
	tyP0400ProdSel.tyProdSel.tyTxtFlippedBrd.uiRtStat.0	:= TRUE;
	tyP0400ProdSel.tyRcpDet.tyTxtFlippedBrd.uiRtStat.0	:= TRUE;

	//Product Selection
	tyP0400ProdSel.tyProdSel.tyStringRecipeNm.sValue		:= p_tyProdRcpCurrRcp0.sRcpNm;
	tyP0400ProdSel.tyProdSel.tyNumProdWidth.diValue			:= p_tyProdRcpCurrRcp0.diWidthInUM;
	tyP0400ProdSel.tyProdSel.tyTxtMcMod.usiValueIdx			:= p_tyProdRcpCurrRcp0.usiMcMod;
	tyP0400ProdSel.tyProdSel.tyTxtFlippedBrd.usiValueIdx	:= p_tyProdRcpCurrRcp0.usiFlippedBrd;
	tyP0400ProdSel.tyProdSel.tyStringMatchCode.sValue		:= p_tyProdRcpCurrRcp0.sMatchCode;

	IF p_tyNtParamCurr.bLFProdWidth2Prep THEN
		fUIInRtStatOff(ADR(tyP0400ProdSel.tyProdSel.tyNumProdWidth2.uiRtStat));
		fUIInRtStatHide(ADR(tyP0400ProdSel.tyProdSel.tyNumProdWidth.uiRtStat));

		fUIInRtStatOff(ADR(tyP0400ProdSel.tyRcpDet.tyNumProdWidth2.uiRtStat));
		fUIInRtStatHide(ADR(tyP0400ProdSel.tyRcpDet.tyNumProdWidth.uiRtStat));

		tyP0400ProdSel.tyProdSel.tyTableRecipe.tyStringTitle2Col2Row0.sValue:= 'US | DS Width';

	ELSE
		fUIInRtStatHide(ADR(tyP0400ProdSel.tyProdSel.tyNumProdWidth2.uiRtStat));
		fUIInRtStatOff(ADR(tyP0400ProdSel.tyProdSel.tyNumProdWidth.uiRtStat));

		fUIInRtStatHide(ADR(tyP0400ProdSel.tyRcpDet.tyNumProdWidth2.uiRtStat));
		fUIInRtStatOff(ADR(tyP0400ProdSel.tyRcpDet.tyNumProdWidth.uiRtStat));

		tyP0400ProdSel.tyProdSel.tyTableRecipe.tyStringTitle2Col2Row0.sValue:= 'Product Width';
	END_IF

END_ACTION
```

#### Act_Main_P0900.st
```iecst
(** 2018-12-21 **)
ACTION Act_Main_P0900:

	//Display
	tyP0900GenIn.tyGenIn.tyBtnCoverSW.uiRtStat.0		:= NOT(p_tyNtParamCurr.tyDISettings.diCoverSWSig > 0);

	tyP0900GenIn.tyGenIn.tyBtnThermalPrtSig.uiRtStat.0	:= NOT(p_tyNtParamCurr.tyDISettings.diThermalPrtSig > 0);
	tyP0900GenIn.tyGenIn.tyBtnPressureSW.uiRtStat.0		:= NOT(p_tyNtParamCurr.tyDISettings.diPressureSW > 0);
	tyP0900GenIn.tyGenIn.tySigLyr.uiRtStat.0			:= NOT(p_tyNtParamCurr.tyDISettings.diThermalPrtSig > 0 OR p_tyNtParamCurr.tyDISettings.diPressureSW > 0);

	tyP0900GenIn.tyGenIn.tyBtnUSWidthChkSen.uiRtStat.0	:= NOT(p_tyNtParamCurr.tyDISettings.diUSWidthChkSen > 0);
	tyP0900GenIn.tyGenIn.tyBtnDSWidthChkSen.uiRtStat.0	:= NOT(p_tyNtParamCurr.tyDISettings.diDSWidthChkSen > 0);
	tyP0900GenIn.tyGenIn.tyWidthChkLyr.uiRtStat.0		:= NOT(p_tyNtParamCurr.tyDISettings.diUSWidthChkSen > 0 OR p_tyNtParamCurr.tyDISettings.diDSWidthChkSen > 0);

	// ADD
	tyP0900GenIn.tyGenIn.tyBtnSafetySigFromDS.uiRtStat := NOT(p_tyNtParamCurr.tyDISettings.diSafetySigFromDS >0 );
	tyP0900GenIn.tyGenIn.tyBtnSafetySigFromUS.uiRtStat := NOT(p_tyNtParamCurr.tyDISettings.diSafetySigFromUS >0 );
	tyP0900GenIn.tyGenIn.tyBtnUlkCoverFromDS.uiRtStat := NOT(p_tyNtParamCurr.tyDISettings.diUnlockCoverSigFromDS >0);
	tyP0900GenIn.tyGenIn.tyBtnUlkCoverFromUS.uiRtStat := NOT(p_tyNtParamCurr.tyDISettings.diUnlockCoverSigFromUS >0);
	tyP0900GenIn.tyGenIn.tyBtnUnlkCovPB.uiRtStat  := NOT(p_tyNtParamCurr.tyDISettings.diCoverUnlockPB1 >0);
	tyP0900GenIn.tyGenIn.tyBtnTopCovSwSIg.uiRtStat := NOT(p_tyNtParamCurr.tyDISettings.diCoverSWSig2 >0);
	tyP0900GenIn.tyGenIn.tyMachSafetyLyr.uiRtStat := NOT(p_tyNtParamCurr.tyDISettings.diSafetySigFromDS >0 OR p_tyNtParamCurr.tyDISettings.diSafetySigFromUS >0  );
END_ACTION
```

#### Act_Main_P0910.st
```iecst
(** 2018-12-21 **)
ACTION Act_Main_P0910:

	//Display
	tyP0910GenOut.tyGenOut.tyBtnBuzzer.uiRtStat.0	:= NOT(p_tyNtParamCurr.tyDOSettings.diBuz > 0);

	tyP0910GenOut.tyGenOut.tyBtnTLGreen.uiRtStat.0	:= NOT(p_tyNtParamCurr.tyDOSettings.diTLGreen > 0);
	tyP0910GenOut.tyGenOut.tyBtnTLAmber.uiRtStat.0	:= NOT(p_tyNtParamCurr.tyDOSettings.diTLAmber > 0);
	tyP0910GenOut.tyGenOut.tyBtnTLRed.uiRtStat.0	:= NOT(p_tyNtParamCurr.tyDOSettings.diTLRed > 0);
	tyP0910GenOut.tyGenOut.tyBtnTLWhite.uiRtStat.0	:= NOT(p_tyNtParamCurr.tyDOSettings.diTLWhite > 0);
	tyP0910GenOut.tyGenOut.tyBtnTLBlue.uiRtStat.0	:= NOT(p_tyNtParamCurr.tyDOSettings.diTLBlue > 0);

	tyP0910GenOut.tyGenOut.tyTLLyr.uiRtStat.0		:= NOT(p_tyNtParamCurr.tyDOSettings.diTLGreen > 0 OR p_tyNtParamCurr.tyDOSettings.diTLAmber > 0 OR p_tyNtParamCurr.tyDOSettings.diTLRed > 0 OR p_tyNtParamCurr.tyDOSettings.diTLWhite > 0 OR p_tyNtParamCurr.tyDOSettings.diTLBlue > 0);
	tyP0910GenOut.tyGenOut.tyBtnTLRed1.uiRtStat.0	:= TRUE;

	//ADD
	tyP0910GenOut.tyGenOut.tyBtnUlkCovPBLED.uiRtStat.0		:= NOT(p_tyNtParamCurr.tyDOSettings.diCoverPBLED1 > 0);
	tyP0910GenOut.tyGenOut.tyBtnTopCovUlkUSDS.uiRtStat.0 	:= NOT(p_tyNtParamCurr.tyDOSettings.diTopCvrUnlckToDS > 0);
	tyP0910GenOut.tyGenOut.tyBtnUlkCovHoldRely.uiRtStat.0:= NOT(p_tyNtParamCurr.tyDOSettings.diBypassTopCover1 > 0);
	tyP0910GenOut.tyGenOut.tyBtnSftSigToUSDS.uiRtStat.0 := NOT(p_tyNtParamCurr.tyDOSettings.diMachineSafetySigToDS > 0);
	tyP0910GenOut.tyGenOut.tyBtnSftUlkCovSWCoil.uiRtStat.0 := NOT(p_tyNtParamCurr.tyDOSettings.diSafetyTopCoverSWCoil1 > 0);

	tyP0910GenOut.tyGenOut.tyUlkCovLyr.uiRtStat.0 := NOT(p_tyNtParamCurr.tyDOSettings.diCoverPBLED1 > 0 OR p_tyNtParamCurr.tyDOSettings.diTopCvrUnlckToDS > 0 OR p_tyNtParamCurr.tyDOSettings.diBypassTopCover1 > 0 );
	tyP0910GenOut.tyGenOut.tyMacSafetyLyr.uiRtStat.0:= NOT(p_tyNtParamCurr.tyDOSettings.diMachineSafetySigToDS > 0 OR p_tyNtParamCurr.tyDOSettings.diSafetyTopCoverSWCoil1 > 0);
END_ACTION
```

#### Act_Main_P0920.st
```iecst
(** 2018-12-21 **)
ACTION Act_Main_P0920:

	//Display
	//Auto-Width
	tyP0920MtrNPneuCtrl.tyMtrNPneuCtrl.tyBtnAW.uiRtStat.0				:= NOT p_tyNtParamCurr.bAWPrep;

	//Stopper
	tyP0920MtrNPneuCtrl.tyMtrNPneuCtrl.tyBtnStopper.uiRtStat.0			:= NOT p_tyNtParamCurr.bProjStopperPrep;

	//Shutter
	tyP0920MtrNPneuCtrl.tyMtrNPneuCtrl.tyBtnShutter.uiRtStat.0			:= NOT (p_tyNtParamCurr.bProjInletShutPrep OR p_tyNtParamCurr.bProjOutletShutPrep);

	//Clamp No RS
	tyP0920MtrNPneuCtrl.tyMtrNPneuCtrl.tyBtnClampNoRS.uiRtStat.0		:= NOT (p_tyNtParamCurr.bProjClampPrep AND (p_tyNtParamCurr.eProjClampOption=ClampNoRS));

	//Clamp With RS
	tyP0920MtrNPneuCtrl.tyMtrNPneuCtrl.tyBtnClampWithRS.uiRtStat.0		:= NOT (p_tyNtParamCurr.bProjClampPrep AND (p_tyNtParamCurr.eProjClampOption=ThreeClampsWithRS));

	IF p_tyNtParamCurr.tyDOSettings.diTLGreen<>0 OR p_tyNtParamCurr.tyDOSettings.diTLAmber<>0 OR p_tyNtParamCurr.tyDOSettings.diTLRed<>0 THEN
		IF p_tyNtParamCurr.eTLBuzMode=TLBuzModBHTC THEN
			tyP0920MtrNPneuCtrl.tyMtrNPneuCtrl.tyBitmapConv.usiValueIdx 	:= 200;
			tyP0920MtrNPneuCtrl.tyMtrNPneuCtrl.tyBitmapShutter.usiValueIdx 	:= 200;
			tyP0920MtrNPneuCtrl.tyMtrNPneuCtrl.tyBitmapAW.usiValueIdx 		:= 200;
		ELSE
			tyP0920MtrNPneuCtrl.tyMtrNPneuCtrl.tyBitmapConv.usiValueIdx 	:= 100;
			tyP0920MtrNPneuCtrl.tyMtrNPneuCtrl.tyBitmapShutter.usiValueIdx 	:= 100;
			tyP0920MtrNPneuCtrl.tyMtrNPneuCtrl.tyBitmapAW.usiValueIdx 		:= 100;
		END_IF
	ELSE
		tyP0920MtrNPneuCtrl.tyMtrNPneuCtrl.tyBitmapConv.usiValueIdx 	:= 0;
		tyP0920MtrNPneuCtrl.tyMtrNPneuCtrl.tyBitmapShutter.usiValueIdx 	:= 0;
		tyP0920MtrNPneuCtrl.tyMtrNPneuCtrl.tyBitmapAW.usiValueIdx 		:= 0;
	END_IF
END_ACTION
```

#### Act_Main_P0922.st
```iecst
ACTION Act_Main_P0922:

	//Display
	tyP0922InletNOutletShutter.tyInletShutterCom.tyLyr.uiRtStat.0	:= NOT(p_tyNtParamCurr.bProjInletShutPrep);
	tyP0922InletNOutletShutter.tyInletShutterDC.tyLyr.uiRtStat.0	:= TRUE;
	tyP0922InletNOutletShutter.tyInletShutterFB.tyLyr.uiRtStat.0	:= NOT(p_tyNtParamCurr.bProjInletShutPrep);

	tyP0922InletNOutletShutter.tyOutletShutterCom.tyLyr.uiRtStat.0	:= NOT(p_tyNtParamCurr.bProjOutletShutPrep);
	tyP0922InletNOutletShutter.tyOutletShutterDC.tyLyr.uiRtStat.0	:= TRUE;
	tyP0922InletNOutletShutter.tyOutletShutterFB.tyLyr.uiRtStat.0	:= NOT(p_tyNtParamCurr.bProjOutletShutPrep);
	tyP0922InletNOutletShutter.tyOutletShutterDis.tyLyr.uiRtStat.0	:= TRUE;

END_ACTION
```

#### Act_Main_P0931.st
```iecst
(** 2018-12-21 **)
ACTION Act_Main_P0931:

	//Display
	tyP0931ConvInv.tyConvCom.tyBtnLft.uiRtStat.0	:= p_tyNtParamCurr.tyDISettings.diConvLftSen = 0;
	tyP0931ConvInv.tyConvCom.tyBtnRgt.uiRtStat.0	:= p_tyNtParamCurr.tyDISettings.diConvRgtSen = 0;

	tyP0931ConvInv.tyInvCom.tyBtnHomeSen.uiRtStat.0	:= p_tyNtParamCurr.tyDISettings.diInvertHomeSen = 0;
	tyP0931ConvInv.tyInvCom.tyBtnRemoteSen.uiRtStat.0	:= p_tyNtParamCurr.tyDISettings.diInvertRemoteSen = 0;

	IF p_tyNtParamCurr.tyDOSettings.diTLGreen<>0 OR p_tyNtParamCurr.tyDOSettings.diTLAmber<>0 OR p_tyNtParamCurr.tyDOSettings.diTLRed<>0 THEN
		IF p_tyNtParamCurr.eTLBuzMode=TLBuzModBHTC THEN
			tyP0931ConvInv.tyConvCom.tyBitmapMc.usiValueIdx := 200;
		ELSE
			tyP0931ConvInv.tyConvCom.tyBitmapMc.usiValueIdx := 100;
		END_IF
	ELSE
		tyP0931ConvInv.tyConvCom.tyBitmapMc.usiValueIdx := 0;
	END_IF

END_ACTION
```

#### Act_Main_P0934.st
```iecst
(** 2018-12-21 **)
ACTION Act_Main_P0934:

	tyP0934AW.tyMotionStd.tyNumTargetPos.diValue	:= 0;
	tyP0934AW.tyMotionStd.tyNumStepSize.diValue		:= 0;
	tyP0934AW.tyMotionStd.tyNumNomSpd.diValue		:= (p_tyNtParamCurr.tyUIAWNomSpd.diMax + p_tyNtParamCurr.tyUIAWNomSpd.diMin) / 2;
	tyP0934AW.tyMotionStd.tyNumSlwSpd.diValue		:= (p_tyNtParamCurr.tyUIAWSlwSpd.diMax + p_tyNtParamCurr.tyUIAWSlwSpd.diMin) / 3;

	tyP0934AW.tyMotionStd.tyNumTargetPos.diValueMax	:= p_tyNtParamCurr.tyProdRcpWidthLmt.diMax;
	tyP0934AW.tyMotionStd.tyNumTargetPos.diValueMin	:= p_tyNtParamCurr.tyUIAWTargetPos.diMin;

	tyP0934AW.tyMotionStd.tyNumStepSize.diValueMax	:= p_tyNtParamCurr.tyProdRcpWidthLmt.diMax;
	tyP0934AW.tyMotionStd.tyNumStepSize.diValueMin	:= p_tyNtParamCurr.tyProdRcpWidthLmt.diMax * -1;

	tyP0934AW.tyMotionStd.tyNumNomSpd.diValueMax	:= p_tyNtParamCurr.tyUIAWNomSpd.diMax;
	tyP0934AW.tyMotionStd.tyNumNomSpd.diValueMin	:= p_tyNtParamCurr.tyUIAWNomSpd.diMin;

	tyP0934AW.tyMotionStd.tyNumSlwSpd.diValueMax	:= p_tyNtParamCurr.tyUIAWSlwSpd.diMax;
	tyP0934AW.tyMotionStd.tyNumSlwSpd.diValueMin	:= p_tyNtParamCurr.tyUIAWSlwSpd.diMin;

	tyP0934AW.tyAW.tyNumNewWidth.diValueMax			:= p_tyNtParamCurr.tyProdRcpWidthLmt.diMax;
	tyP0934AW.tyAW.tyNumNewWidth.diValueMin			:= p_tyNtParamCurr.tyProdRcpWidthLmt.diMin;

END_ACTION
```

#### Act_Main_P0940.st
```iecst
ACTION Act_Main_P0940:

	//Display
	tyP0940CommCtrl.tyUSSMEMA2.tyLyr.uiRtStat.0	:= NOT(p_tyNtParamCurr.bProjInvertOncePrep  OR p_tyNtParamCurr.bProjInvertTwicePrep);

	tyP0940CommCtrl.tyUSSMEMA.tyBtnUBA.uiRtStat.0		:= p_tyNtParamCurr.tyDISettings.diUBA = 0;
	tyP0940CommCtrl.tyUSSMEMA.tyBtnUBAStat.uiRtStat.0	:= p_tyNtParamCurr.tyDISettings.diUBAStat = 0;
	tyP0940CommCtrl.tyUSSMEMA.tyBtnUSB.uiRtStat.0		:= p_tyNtParamCurr.tyDOSettings.diUSB = 0;

	tyP0940CommCtrl.tyDSSMEMA.tyBtnDSB.uiRtStat.0		:= p_tyNtParamCurr.tyDISettings.diDSB = 0;
	tyP0940CommCtrl.tyDSSMEMA.tyBtnDBA.uiRtStat.0		:= p_tyNtParamCurr.tyDOSettings.diDBA = 0;
	tyP0940CommCtrl.tyDSSMEMA.tyBtnDBAStat.uiRtStat.0	:= p_tyNtParamCurr.tyDOSettings.diDBAStat = 0;

	tyP0940CommCtrl.tyUSSMEMA2.tyBtnUBA.uiRtStat.0		:= p_tyNtParamCurr.tyDISettings.diUBA2 = 0;
	tyP0940CommCtrl.tyUSSMEMA2.tyBtnUBAStat.uiRtStat.0	:= p_tyNtParamCurr.tyDISettings.diUBAStat2 = 0;
	tyP0940CommCtrl.tyUSSMEMA2.tyBtnUSB.uiRtStat.0		:= p_tyNtParamCurr.tyDOSettings.diUSB2 = 0;

END_ACTION
```

#### Act_Main_P1000.st
```iecst
(** 2018-12-21 **)
ACTION Act_Main_P1000:

	//Language
	p_tyMcParamCurr.usiLang	:= 0;

//	fUIInRtStatHide(ADR(tyP1000Lang.tyLang.tyBtnGerman.uiRtStat));
//	fUIInRtStatHide(ADR(tyP1000Lang.tyLang.tyBtnChinese.uiRtStat));

//	CASE p_tyMcParamCurr.usiLang OF
//		1:
//			tyP1000Lang.tyLang.tyBtnEnglish.bValue	:= FALSE;
//			tyP1000Lang.tyLang.tyBtnEnglish.bRtLk	:= FALSE;
//			tyP1000Lang.tyLang.tyBtnGerman.bValue	:= TRUE;
//			tyP1000Lang.tyLang.tyBtnGerman.bRtLk	:= TRUE;
//			tyP1000Lang.tyLang.tyBtnChinese.bValue	:= FALSE;
//			tyP1000Lang.tyLang.tyBtnChinese.bRtLk	:= FALSE;
//		2:
//			tyP1000Lang.tyLang.tyBtnEnglish.bValue	:= FALSE;
//			tyP1000Lang.tyLang.tyBtnEnglish.bRtLk	:= FALSE;
//			tyP1000Lang.tyLang.tyBtnGerman.bValue	:= FALSE;
//			tyP1000Lang.tyLang.tyBtnGerman.bRtLk	:= FALSE;
//			tyP1000Lang.tyLang.tyBtnChinese.bValue	:= TRUE;
//			tyP1000Lang.tyLang.tyBtnChinese.bRtLk	:= TRUE;
//		ELSE
//			tyP1000Lang.tyLang.tyBtnEnglish.bValue	:= TRUE;
//			tyP1000Lang.tyLang.tyBtnEnglish.bRtLk	:= TRUE;
//			tyP1000Lang.tyLang.tyBtnGerman.bValue	:= FALSE;
//			tyP1000Lang.tyLang.tyBtnGerman.bRtLk	:= FALSE;
//			tyP1000Lang.tyLang.tyBtnChinese.bValue	:= FALSE;
//			tyP1000Lang.tyLang.tyBtnChinese.bRtLk	:= FALSE;
//	END_CASE

END_ACTION
```

#### Act_Main_P1020.st
```iecst
ACTION Act_Main_P1020:

	//Display
	tyP1020McSetNavi.tyNavi.tyBtnVCommSet.uiRtStat.0	:= NOT(p_tyNtParamCurr.bLFPrep OR p_tyNtParamCurr.bLCSLFPrep OR p_tyNtParamCurr.bLCSReqRcpPrep OR p_tyNtParamCurr.bLCSLiveDatPrep);

END_ACTION
```

#### Act_Main_P1021.st
```iecst
(** 2018-12-21 **)
ACTION Act_Main_P1021:

	//Machine Setting_General
	tyP1021McSetGen.tyGen.tyNumConvInitTm.diValueMin	:= p_tyNtParamCurr.tyUIConvInitTm.diMin;
	tyP1021McSetGen.tyGen.tyNumConvInitTm.diValueMax	:= p_tyNtParamCurr.tyUIConvInitTm.diMax;

	tyP1021McSetGen.tyGen.tyNumTranInErrDlyTm.diValueMin	:= p_tyNtParamCurr.tyUITranInErrDlyTm.diMin;
	tyP1021McSetGen.tyGen.tyNumTranInErrDlyTm.diValueMax	:= p_tyNtParamCurr.tyUITranInErrDlyTm.diMax;

	tyP1021McSetGen.tyGen.tyNumTranOutErrDlyTm.diValueMin	:= p_tyNtParamCurr.tyUITranOutErrDlyTm.diMin;
	tyP1021McSetGen.tyGen.tyNumTranOutErrDlyTm.diValueMax	:= p_tyNtParamCurr.tyUITranOutErrDlyTm.diMax;

	tyP1021McSetGen.tyGen.tyDrpDnDefaultMcMod.usiValueMinIdx	:= DINT_TO_USINT(p_tyNtParamCurr.tyProdRcpMcModLmt.diMin);
	tyP1021McSetGen.tyGen.tyDrpDnDefaultMcMod.usiValueMaxIdx	:= DINT_TO_USINT(p_tyNtParamCurr.tyProdRcpMcModLmt.diMax);

	//Network Mode
	tyP1021McSetGen.tyGen.tyDrpDnNetworkMod.usiValueMinIdx		:= DINT_TO_USINT(p_tyNtParamCurr.tyNetworkMode.diMin);
	tyP1021McSetGen.tyGen.tyDrpDnNetworkMod.usiValueMaxIdx		:= DINT_TO_USINT(p_tyNtParamCurr.tyNetworkMode.diMax);

	tyP1021McSetGen.tyGen.tyDrpDnDefaultFlippedBrd.usiValueMinIdx	:= DINT_TO_USINT(p_tyNtParamCurr.tyProdRcpFlippedBrdLmt.diMin);
	tyP1021McSetGen.tyGen.tyDrpDnDefaultFlippedBrd.usiValueMaxIdx	:= DINT_TO_USINT(p_tyNtParamCurr.tyProdRcpFlippedBrdLmt.diMax);

	tyP1021McSetGen.tyGen.tyNumStopperAtLftPos.diValueMin	:= p_tyNtParamCurr.tyUIInvertTargetPos.diMin;
	tyP1021McSetGen.tyGen.tyNumStopperAtLftPos.diValueMax	:= p_tyNtParamCurr.tyUIInvertTargetPos.diMax;
	tyP1021McSetGen.tyGen.tyNumStopperAtRgtPos.diValueMin	:= p_tyNtParamCurr.tyUIInvertTargetPos.diMin;
	tyP1021McSetGen.tyGen.tyNumStopperAtRgtPos.diValueMax	:= p_tyNtParamCurr.tyUIInvertTargetPos.diMax;

	//Screen Saver
	tyP1021McSetGen.tyGen.tyNumSSaverTm.diValueMin			:= p_tyNtParamCurr.tyUISSaverTm.diMin;
	tyP1021McSetGen.tyGen.tyNumSSaverTm.diValueMax			:= p_tyNtParamCurr.tyUISSaverTm.diMax;
	tyP1021McSetGen.tyGen.tyNumSSaverTm.uiRtStat.0			:= NOT p_tyNtParamCurr.bSSaverPrep;
	tyP1021McSetGen.tyGen.tyTxtSSaverTm.uiRtStat.0			:= NOT p_tyNtParamCurr.bSSaverPrep;
	tyP1021McSetGen.tyGen.tyBtnSSaverEn.uiRtStat.0			:= NOT p_tyNtParamCurr.bSSaverPrep;

	//Logout
	tyP1021McSetGen.tyGen.tyNumAutoLogoutTm.diValueMin			:= p_tyNtParamCurr.tyUIAutoLogoutTm.diMin;
	tyP1021McSetGen.tyGen.tyNumAutoLogoutTm.diValueMax			:= p_tyNtParamCurr.tyUIAutoLogoutTm.diMax;
	tyP1021McSetGen.tyGen.tyNumAutoLogoutTm.uiRtStat.0			:= NOT p_tyNtParamCurr.bAutoLogoutPrep;
	tyP1021McSetGen.tyGen.tyTxtLblAutoLogoutTm.uiRtStat.0		:= NOT p_tyNtParamCurr.bAutoLogoutPrep;
	tyP1021McSetGen.tyGen.tyBtnAutoLogoutEn.uiRtStat.0			:= NOT p_tyNtParamCurr.bAutoLogoutPrep;

	//Width
	tyP1021McSetGen.tyGen.tyNumWidthAtHm.diValueMin			:= p_tyNtParamCurr.tyProdRcpWidthLmt.diMin;
	tyP1021McSetGen.tyGen.tyNumWidthAtHm.diValueMax			:= p_tyNtParamCurr.tyProdRcpWidthLmt.diMax + 10000;
	tyP1021McSetGen.tyGen.tyNumWidthAtHm.uiRtStat.0			:= NOT p_tyNtParamCurr.bAWPrep;
	tyP1021McSetGen.tyGen.tyTxtWidthAtHm.uiRtStat.0			:= NOT p_tyNtParamCurr.bAWPrep;
	tyP1021McSetGen.tyGen.tyBtnAWDis.uiRtStat.0				:= NOT p_tyNtParamCurr.bAWPrep;

	//Width Offset
	//tyP1021McSetGen.tyGen.tyNumWidthOffset.uiRtStat.0		:= NOT p_tyNtParamCurr.bAWPrep;
	//tyP1021McSetGen.tyGen.tyTxtWidthOffset.uiRtStat.0		:= NOT p_tyNtParamCurr.bAWPrep;
	tyP1021McSetGen.tyGen.tyNumWidthOffset.uiRtStat.0		:= TRUE;
	tyP1021McSetGen.tyGen.tyTxtWidthOffset.uiRtStat.0		:= TRUE;
	tyP1021McSetGen.tyGen.tyNumWidthOffset.diValueMin		:= p_tyNtParamCurr.tyUIAWOffset.diMin;
	tyP1021McSetGen.tyGen.tyNumWidthOffset.diValueMax		:= p_tyNtParamCurr.tyUIAWOffset.diMax;

	//Virtual SMEMA
	tyP1021McSetGen.tyGen.tyBtnVSMEMAEn.uiRtStat.0	:= NOT p_tyNtParamCurr.bVSMEMAPrep;

	//Hermes Remote Configuration
	tyP1021McSetGen.tyGen.tyBtnHermesRmtEn.uiRtStat.0	:= NOT p_tyNtParamCurr.bHermesRmtPrep;

	//Stopper
	//tyP1021McSetGen.tyGen.tyBtnStopperDis.uiRtStat.0	:= NOT p_tyNtParamCurr.bProjStopperPrep;
	tyP1021McSetGen.tyGen.tyBtnStopperDis.uiRtStat.0	:= TRUE;

	//Stopper
	tyP1021McSetGen.tyGen.tyBtnClampDis.uiRtStat.0	:= NOT (p_tyNtParamCurr.bProjClampPrep AND (p_tyNtParamCurr.eProjClampOption=ClampNoRS));

	//Display Flipped Board
	tyP1021McSetGen.tyGen.tyTxtLblFlippedBrd.uiRtStat.0	:= TRUE;
	tyP1021McSetGen.tyGen.tyDrpDnDefaultFlippedBrd.uiRtStat.0 :=TRUE;

	//Parameter
	tyP1021McSetGen.tyGen.tyStringMcNm.sValue					:= p_tyMcParamCurr.sMcNm;
	tyP1021McSetGen.tyGen.tyNumWidthAtHm.diValue				:= p_tyMcParamCurr.diWidthAtHmPosInUM;
	tyP1021McSetGen.tyGen.tyStringIPAddr.sValue					:= p_sHWInfoIPAddr;
	tyP1021McSetGen.tyGen.tyStringSubnetMask.sValue				:= p_sHWInfoSubnetMask;
	tyP1021McSetGen.tyGen.tyNumSSaverTm.diValue					:= UINT_TO_DINT(p_tyMcParamCurr.uiSSaverTmInSec);
	tyP1021McSetGen.tyGen.tyBtnSSaverEn.bValue					:= p_tyMcParamCurr.bSSaverEn;

	tyP1021McSetGen.tyGen.tyNumConvInitTm.diValue				:= p_tyMcParamCurr.diConvInitTmInMS;
	tyP1021McSetGen.tyGen.tyNumTranInErrDlyTm.diValue			:= p_tyMcParamCurr.diTranInErrDlyTmInMS;
	tyP1021McSetGen.tyGen.tyNumTranOutErrDlyTm.diValue			:= p_tyMcParamCurr.diTranOutErrDlyTmInMS;
	tyP1021McSetGen.tyGen.tyDrpDnDefaultMcMod.usiValueIdx		:= p_tyMcParamCurr.usiDefaultMcMod;
	tyP1021McSetGen.tyGen.tyDrpDnDefaultFlippedBrd.usiValueIdx	:= p_tyMcParamCurr.usiDefaultFlippedBrd;

	tyP1021McSetGen.tyGen.tyBtnAutoStepEn.bValue				:= p_tyMcParamCurr.bAutoStepEn;
	tyP1021McSetGen.tyGen.tyBtnAWDis.bValue						:= p_tyMcParamCurr.bAWDis;
	tyP1021McSetGen.tyGen.tyBtnVSMEMAEn.bValue					:= p_tyMcParamCurr.bVSMEMAEn;
	tyP1021McSetGen.tyGen.tyBtnMnlAccDat.bValue					:= p_tyMcParamCurr.bMnlAccDat;
	tyP1021McSetGen.tyGen.tyBtnChgParamEn.bValue				:= p_tyMcParamCurr.bChgParamEn;
	tyP1021McSetGen.tyGen.tyBtnHermesRmtEn.bValue				:= p_tyMcParamCurr.bHermesRmtEn;

	tyP1021McSetGen.tyGen.tyBtnStopperDis.bValue				:= p_tyMcParamCurr.bStopperDis;
	tyP1021McSetGen.tyGen.tyNumStopperAtLftPos.diValue			:= p_tyMcParamCurr.diStopperAtLftPos;
	tyP1021McSetGen.tyGen.tyNumStopperAtRgtPos.diValue			:= p_tyMcParamCurr.diStopperAtRgtPos;

	tyP1021McSetGen.tyGen.tyNumAutoLogoutTm.diValue				:= p_tyMcParamCurr.diAutoLogoutTmInSec;
	tyP1021McSetGen.tyGen.tyBtnAutoLogoutEn.bValue				:= p_tyMcParamCurr.bAutoLogoutEn;

	tyP1021McSetGen.tyGen.tyBtnClampDis.bValue					:= p_tyMcParamCurr.bClampDis;

	tyP1021McSetGen.tyGen.tyDrpDnNetworkMod.usiValueIdx		:= DINT_TO_USINT(p_tyMcParamCurr.eNetworkMod);
	tyP1021McSetGen.tyGen.tyBtnLFBuzMute.bValue				:= p_tyMcParamCurr.bLFBuzMute;

	tyP1021McSetGen.tyGen.tyBtnAutoStepEn.uiRtStat.0			:= TRUE;
END_ACTION
```

#### Act_Main_P1022.st
```iecst
ACTION Act_Main_P1022:

	//Machine Setting - Vertical Communicationm Control
	//Display
	tyP1022McSetVComm.tyVComSel.tyBtnLF.uiRtStat.0				:= NOT p_tyNtParamCurr.bLFPrep;
	tyP1022McSetVComm.tyVComSel.tyBtnLCSLF.uiRtStat.0			:= NOT p_tyNtParamCurr.bLCSLFPrep;
	tyP1022McSetVComm.tyVComSel.tyBtnLCSReqRcp.uiRtStat.0		:= NOT p_tyNtParamCurr.bLCSReqRcpPrep;
	tyP1022McSetVComm.tyVComSel.tyBtnLCSManageRcp.uiRtStat.0	:= NOT p_tyNtParamCurr.bLCSManageRcpPrep;
	tyP1022McSetVComm.tyVComSel.tyBtnLCSLiveDat.uiRtStat.0		:= NOT p_tyNtParamCurr.bLCSLiveDatPrep;

	tyP1022McSetVComm.tyLF.tyBtnLeaderMc.uiRtStat.0				:= NOT p_tyNtParamCurr.bLFUsrSetPrep;
//	tyP1022McSetVComm.tyLF.tyBtnSectionLdr.uiRtStat.0			:= NOT p_tyNtParamCurr.bLFPrep OR NOT p_tyNtParamCurr.bLCSLFPrep;
	tyP1022McSetVComm.tyLF.tyBtnUSWidthChkEn.uiRtStat.0			:= NOT p_tyNtParamCurr.bUSWidthChkPrep;
	tyP1022McSetVComm.tyLF.tyBtnDSWidthChkEn.uiRtStat.0			:= NOT p_tyNtParamCurr.bDSWidthChkPrep;
	tyP1022McSetVComm.tyLF.tyBtnSeqStayActive.uiRtStat.0		:= TRUE ;
	tyP1022McSetVComm.tyLF.tyBtnDBAOnWOAlign.uiRtStat.0			:= NOT p_tyNtParamCurr.bDSWidthChkPrep;

	//Parameter
	tyP1022McSetVComm.tyVComSel.tyBtnLF.bValue					:= p_tyMcParamCurr.bLFEn;
	tyP1022McSetVComm.tyVComSel.tyBtnLCSLF.bValue				:= p_tyMcParamCurr.bLCSLFEn;
	tyP1022McSetVComm.tyVComSel.tyBtnLCSReqRcp.bValue			:= p_tyMcParamCurr.bLCSReqRcpEn;
	tyP1022McSetVComm.tyVComSel.tyBtnLCSManageRcp.bValue		:= p_tyMcParamCurr.bLCSManageRcpEn;
	tyP1022McSetVComm.tyVComSel.tyBtnLCSLiveDat.bValue			:= p_tyMcParamCurr.bLCSLiveDatEn;

	tyP1022McSetVComm.tyLF.tyBtnLeaderMc.bValue					:= p_tyMcParamCurr.bLFLeaderMc;
	tyP1022McSetVComm.tyLF.tyBtnSectionLdr.bValue				:= p_tyMcParamCurr.bSectionLeader;
	tyP1022McSetVComm.tyLF.tyBtnUSWidthChkEn.bValue				:= p_tyMcParamCurr.bUSWidthChkEn;
	tyP1022McSetVComm.tyLF.tyBtnDSWidthChkEn.bValue				:= p_tyMcParamCurr.bDSWidthChkEn;
	tyP1022McSetVComm.tyLF.tyBtnSeqStayActive.bValue			:= p_tyMcParamCurr.bLFSeqStayActive;
	tyP1022McSetVComm.tyLF.tyBtnDBAOnWOAlign.bValue				:= p_tyMcParamCurr.bDBAOnWOAlign;

	//new for Hermes 1.3
	tyP1022McSetVComm.tyVComSvy.tyNumSndAliveTm.diValue	    	    := TIME_TO_DINT(p_tyHermesConfiguration.tySvyParam.tSndAlive);
	tyP1022McSetVComm.tyVComSvy.tyNumSvySystemPort.diValue	    	:= UINT_TO_DINT(p_tyHermesConfiguration.tySvyParam.uiSvySvstemPort);
	tyP1022McSetVComm.tyVComSvy.tyBtnConfiguration.bValue		    := p_tyHermesConfiguration.tySvyParam.bFeatureConfiguration;
	tyP1022McSetVComm.tyVComSvy.tyBtnCheckAliveResponse.bValue		:= p_tyHermesConfiguration.tySvyParam.bFeatureCheckAliveResponse;
	tyP1022McSetVComm.tyVComSvy.tyBtnBoardTracking.bValue		    := p_tyHermesConfiguration.tySvyParam.bFeatureBoardTracking;
	tyP1022McSetVComm.tyVComSvy.tyBtnQueryWorkOrderInfo.bValue		:= p_tyHermesConfiguration.tySvyParam.bFeatureQueryWorkOrderInfo;
	tyP1022McSetVComm.tyVComSvy.tyBtnSendWorkOrderInfo.bValue		:= p_tyHermesConfiguration.tySvyParam.bFeatureSendWorkOrderInfo;

	//Hermes 1.3 Board Reinsert Function
	tyP1022McSetVComm.tyVComSvy.tyBtnInsertBrd.bValue		:= p_tyHermesConfiguration.tySvyParam.bFeatureInsertBrd;
END_ACTION
```

#### Act_Main_P1023.st
```iecst
(** 2018-12-21 **)
ACTION Act_Main_P1023:

	//Machine Setting_Communicationm Control
	//Display
	tyP1023McSetHComm.tyUSSel.tyBtnHermes.uiRtStat.0	:= NOT p_tyNtParamCurr.bHermesPrep;
	tyP1023McSetHComm.tyDSSel.tyBtnHermes.uiRtStat.0	:= NOT p_tyNtParamCurr.bHermesPrep;

	tyP1023McSetHComm.tyUSSel2.tyBtnHermes.uiRtStat.0	:= NOT (p_tyNtParamCurr.bHermesPrep AND (p_tyNtParamCurr.bProjInvertOncePrep OR p_tyNtParamCurr.bProjInvertTwicePrep)) ;

	IF p_tyNtParamCurr.bUSExtSMEMAPrep = TRUE THEN
		tyP1023McSetHComm.tyUSSMEMA.tyDrpDnSMEMAMod.usiValueMaxIdx	:= 2;

	ELSIF p_tyNtParamCurr.bUSExtSMEMA2Prep = TRUE THEN
		tyP1023McSetHComm.tyUSSMEMA2.tyDrpDnSMEMAMod.usiValueMaxIdx	:= 2;
	ELSE
		tyP1023McSetHComm.tyUSSMEMA.tyDrpDnSMEMAMod.usiValueMaxIdx	:= 1;
		tyP1023McSetHComm.tyUSSMEMA2.tyDrpDnSMEMAMod.usiValueMaxIdx	:= 1;
	END_IF

	IF p_tyNtParamCurr.bDSExtSMEMAPrep = TRUE THEN
		tyP1023McSetHComm.tyDSSMEMA.tyDrpDnSMEMAMod.usiValueMaxIdx	:= 2;
	ELSE
		tyP1023McSetHComm.tyDSSMEMA.tyDrpDnSMEMAMod.usiValueMaxIdx	:= 1;
	END_IF

	//Parameter
	//Upstream
	CASE p_tyMcParamCurr.eUSComm OF
		McSetCommModSMEMA:
			tyP1023McSetHComm.tyUSSel.tyBtnSMEMA.bValue		:= TRUE;
			tyP1023McSetHComm.tyUSSel.tyBtnSMEMA.bRtLk		:= TRUE;
			tyP1023McSetHComm.tyUSSel.tyBtnHermes.bValue	:= FALSE;
			tyP1023McSetHComm.tyUSSel.tyBtnHermes.bRtLk		:= FALSE;
		McSetCommModHermes:
			tyP1023McSetHComm.tyUSSel.tyBtnSMEMA.bValue		:= FALSE;
			tyP1023McSetHComm.tyUSSel.tyBtnSMEMA.bRtLk		:= FALSE;
			tyP1023McSetHComm.tyUSSel.tyBtnHermes.bValue	:= TRUE;
			tyP1023McSetHComm.tyUSSel.tyBtnHermes.bRtLk		:= TRUE;
	END_CASE

	tyP1023McSetHComm.tyUSSMEMA.tyDrpDnSMEMAMod.usiValueIdx		:= UDINT_TO_USINT(p_tyMcParamCurr.tyUSCommSMEMA.eSelection);
	tyP1023McSetHComm.tyUSSMEMA.tyBtnGdSig.bValue				:= p_tyMcParamCurr.tyUSCommSMEMA.bStatSigSetGd;

	tyP1023McSetHComm.tyUSHermes.tyNumSndAliveTm.diValue		:= TIME_TO_DINT(p_tyHermesConfiguration.a_tyUSParam[0].tSndAlive);
	tyP1023McSetHComm.tyUSHermes.tyNumLaneID.diValue			:= INT_TO_DINT(p_tyHermesConfiguration.a_tyUSParam[0].iLaneID);
	tyP1023McSetHComm.tyUSHermes.tyNumHostPort.diValue			:= UINT_TO_DINT(p_tyHermesConfiguration.a_tyUSParam[0].uiHostPort);
	tyP1023McSetHComm.tyUSHermes.tyStringHostAddr.sValue		:= p_tyHermesConfiguration.a_tyUSParam[0].sHostAddress;
	tyP1023McSetHComm.tyUSHermes.tyBtnCheckAliveResponse.bValue	:= p_tyHermesConfiguration.a_tyUSParam[0].bFeatureCheckAliveResponse;
	tyP1023McSetHComm.tyUSHermes.tyBtnBoardForecast.bValue			:= p_tyHermesConfiguration.a_tyUSParam[0].bFeatureBoardForecast;
	tyP1023McSetHComm.tyUSHermes.tyBtnQueryBoardInfo.bValue			:= p_tyHermesConfiguration.a_tyUSParam[0].bFeatureQueryBoardInfo;
	tyP1023McSetHComm.tyUSHermes.tyBtnCommand.bValue			:= p_tyHermesConfiguration.a_tyUSParam[0].bFeatureCommand;

	tyP1023McSetHComm.tyUSHermes.tyBtnCmpTypeId.bValue			:= p_tyHermesConfiguration.a_tyUSParam[0].bCmpTypeId;
	tyP1023McSetHComm.tyUSHermes.tyBtnCmpParam.bValue			:= p_tyHermesConfiguration.a_tyUSParam[0].bCmpParam;
	tyP1023McSetHComm.tyUSHermes.tyBtnOverWrite.bValue			:= p_tyHermesConfiguration.a_tyUSParam[0].bOverwrite;

	//Upstream 2
	CASE p_tyMcParamCurr.eUSComm2 OF
		McSetCommModSMEMA:
			tyP1023McSetHComm.tyUSSel2.tyBtnSMEMA.bValue	:= TRUE;
			tyP1023McSetHComm.tyUSSel2.tyBtnSMEMA.bRtLk		:= TRUE;
			tyP1023McSetHComm.tyUSSel2.tyBtnHermes.bValue	:= FALSE;
			tyP1023McSetHComm.tyUSSel2.tyBtnHermes.bRtLk	:= FALSE;
		McSetCommModHermes:
			tyP1023McSetHComm.tyUSSel2.tyBtnSMEMA.bValue	:= FALSE;
			tyP1023McSetHComm.tyUSSel2.tyBtnSMEMA.bRtLk		:= FALSE;
			tyP1023McSetHComm.tyUSSel2.tyBtnHermes.bValue	:= TRUE;
			tyP1023McSetHComm.tyUSSel2.tyBtnHermes.bRtLk	:= TRUE;
	END_CASE

	tyP1023McSetHComm.tyUSSMEMA2.tyDrpDnSMEMAMod.usiValueIdx	:= UDINT_TO_USINT(p_tyMcParamCurr.tyUSCommSMEMA2.eSelection);
	tyP1023McSetHComm.tyUSSMEMA2.tyBtnGdSig.bValue				:= p_tyMcParamCurr.tyUSCommSMEMA2.bStatSigSetGd;

	tyP1023McSetHComm.tyUSHermes2.tyNumSndAliveTm.diValue		:= TIME_TO_DINT(p_tyHermesConfiguration.a_tyUSParam[1].tSndAlive);
	tyP1023McSetHComm.tyUSHermes2.tyNumLaneID.diValue			:= INT_TO_DINT(p_tyHermesConfiguration.a_tyUSParam[1].iLaneID);
	tyP1023McSetHComm.tyUSHermes2.tyNumHostPort.diValue			:= UINT_TO_DINT(p_tyHermesConfiguration.a_tyUSParam[1].uiHostPort);
	tyP1023McSetHComm.tyUSHermes2.tyStringHostAddr.sValue		:= p_tyHermesConfiguration.a_tyUSParam[1].sHostAddress;
	tyP1023McSetHComm.tyUSHermes2.tyBtnCheckAliveResponse.bValue	:= p_tyHermesConfiguration.a_tyUSParam[1].bFeatureCheckAliveResponse;
	tyP1023McSetHComm.tyUSHermes2.tyBtnBoardForecast.bValue			:= p_tyHermesConfiguration.a_tyUSParam[1].bFeatureBoardForecast;
	tyP1023McSetHComm.tyUSHermes2.tyBtnQueryBoardInfo.bValue			:= p_tyHermesConfiguration.a_tyUSParam[1].bFeatureQueryBoardInfo;
	tyP1023McSetHComm.tyUSHermes2.tyBtnCommand.bValue			:= p_tyHermesConfiguration.a_tyUSParam[1].bFeatureCommand;

	tyP1023McSetHComm.tyUSHermes2.tyBtnCmpTypeId.bValue			:= p_tyHermesConfiguration.a_tyUSParam[1].bCmpTypeId;
	tyP1023McSetHComm.tyUSHermes2.tyBtnCmpParam.bValue			:= p_tyHermesConfiguration.a_tyUSParam[1].bCmpParam;
	tyP1023McSetHComm.tyUSHermes2.tyBtnOverWrite.bValue			:= p_tyHermesConfiguration.a_tyUSParam[1].bOverwrite;

	//Downstream
	CASE p_tyMcParamCurr.eDSComm OF
		McSetCommModSMEMA:
			tyP1023McSetHComm.tyDSSel.tyBtnSMEMA.bValue		:= TRUE;
			tyP1023McSetHComm.tyDSSel.tyBtnSMEMA.bRtLk		:= TRUE;
			tyP1023McSetHComm.tyDSSel.tyBtnHermes.bValue	:= FALSE;
			tyP1023McSetHComm.tyDSSel.tyBtnHermes.bRtLk		:= FALSE;
		McSetCommModHermes:
			tyP1023McSetHComm.tyDSSel.tyBtnSMEMA.bValue		:= FALSE;
			tyP1023McSetHComm.tyDSSel.tyBtnSMEMA.bRtLk		:= FALSE;
			tyP1023McSetHComm.tyDSSel.tyBtnHermes.bValue	:= TRUE;
			tyP1023McSetHComm.tyDSSel.tyBtnHermes.bRtLk		:= TRUE;
	END_CASE

	tyP1023McSetHComm.tyDSSMEMA.tyDrpDnSMEMAMod.usiValueIdx		:= UDINT_TO_USINT(p_tyMcParamCurr.tyDSCommSMEMA.eSelection);
	tyP1023McSetHComm.tyDSSMEMA.tyBtnGdSig.bValue				:= p_tyMcParamCurr.tyDSCommSMEMA.bStatSigSetGd;

	tyP1023McSetHComm.tyDSHermes.tyNumSndAliveTm.diValue		:= TIME_TO_DINT(p_tyHermesConfiguration.a_tyDSParam[0].tSndAlive);
	tyP1023McSetHComm.tyDSHermes.tyNumSvrPort.diValue			:= UINT_TO_DINT(p_tyHermesConfiguration.a_tyDSParam[0].uiSvrPort);
	tyP1023McSetHComm.tyDSHermes.tyNumLaneID.diValue			:= INT_TO_DINT(p_tyHermesConfiguration.a_tyDSParam[0].iLaneID);
	tyP1023McSetHComm.tyDSHermes.tyBtnCheckAliveResponse.bValue	:= p_tyHermesConfiguration.a_tyDSParam[0].bFeatureCheckAliveResponse;
	tyP1023McSetHComm.tyDSHermes.tyBtnBoardForecast.bValue		:= p_tyHermesConfiguration.a_tyDSParam[0].bFeatureBoardForecast;
	tyP1023McSetHComm.tyDSHermes.tyBtnSendBoardInfo.bValue		:= p_tyHermesConfiguration.a_tyDSParam[0].bFeatureSendBoardInfo;
	tyP1023McSetHComm.tyDSHermes.tyBtnCommand.bValue			:= p_tyHermesConfiguration.a_tyDSParam[0].bFeatureCommand;

	//DS 2
	CASE p_tyMcParamCurr.eDSComm2 OF
		McSetCommModSMEMA:
			tyP1023McSetHComm.tyDSSel2.tyBtnSMEMA.bValue		:= TRUE;
			tyP1023McSetHComm.tyDSSel2.tyBtnSMEMA.bRtLk		:= TRUE;
			tyP1023McSetHComm.tyDSSel2.tyBtnHermes.bValue	:= FALSE;
			tyP1023McSetHComm.tyDSSel2.tyBtnHermes.bRtLk		:= FALSE;
		McSetCommModHermes:
			tyP1023McSetHComm.tyDSSel2.tyBtnSMEMA.bValue		:= FALSE;
			tyP1023McSetHComm.tyDSSel2.tyBtnSMEMA.bRtLk		:= FALSE;
			tyP1023McSetHComm.tyDSSel2.tyBtnHermes.bValue	:= TRUE;
			tyP1023McSetHComm.tyDSSel2.tyBtnHermes.bRtLk		:= TRUE;
	END_CASE
	tyP1023McSetHComm.tyDSSMEMA2.tyDrpDnSMEMAMod.usiValueIdx		:= UDINT_TO_USINT(p_tyMcParamCurr.tyDSCommSMEMA2.eSelection);
	tyP1023McSetHComm.tyDSSMEMA2.tyBtnGdSig.bValue				:= p_tyMcParamCurr.tyDSCommSMEMA2.bStatSigSetGd;

	tyP1023McSetHComm.tyDSHermes2.tyNumSndAliveTm.diValue		:= TIME_TO_DINT(p_tyHermesConfiguration.a_tyDSParam[1].tSndAlive);
	tyP1023McSetHComm.tyDSHermes2.tyNumSvrPort.diValue			:= UINT_TO_DINT(p_tyHermesConfiguration.a_tyDSParam[1].uiSvrPort);
	tyP1023McSetHComm.tyDSHermes2.tyNumLaneID.diValue			:= INT_TO_DINT(p_tyHermesConfiguration.a_tyDSParam[1].iLaneID);
	tyP1023McSetHComm.tyDSHermes2.tyBtnCheckAliveResponse.bValue	:= p_tyHermesConfiguration.a_tyDSParam[1].bFeatureCheckAliveResponse;
	tyP1023McSetHComm.tyDSHermes2.tyBtnBoardForecast.bValue		:= p_tyHermesConfiguration.a_tyDSParam[1].bFeatureBoardForecast;
	tyP1023McSetHComm.tyDSHermes2.tyBtnSendBoardInfo.bValue		:= p_tyHermesConfiguration.a_tyDSParam[1].bFeatureSendBoardInfo;
	tyP1023McSetHComm.tyDSHermes2.tyBtnCommand.bValue			:= p_tyHermesConfiguration.a_tyDSParam[1].bFeatureCommand;

	//Upstream Downstream Selection
	tyP1023McSetHComm.tyGen.tyDrpDnUSSel.usiValueIdx 	:= 0;
	tyP1023McSetHComm.tyGen.tyDrpDnDSSel.usiValueIdx	:= 0;

	tyP1023McSetHComm.tyGen.tyDrpDnDSSel.uiRtStat.0				:= NOT (p_tyNtParamCurr.bProjInvertOncePrep AND p_tyNtParamCurr.bProjInvertTwicePrep);
	tyP1023McSetHComm.tyGen.tyDrpDnUSSel.uiRtStat.0				:= NOT (p_tyNtParamCurr.bProjInvertOncePrep AND p_tyNtParamCurr.bProjInvertTwicePrep);

END_ACTION
```

#### Act_Main_P1024.st
```iecst
(** 2018-12-21 **)
ACTION Act_Main_P1024:

	//Display
	IF p_tyNtParamCurr.tyDISettings.diConvLftSen = 0 THEN
		fUIInRtStatHide(ADR(tyP1024McSetAntiGap.tyAntiGap.tyTxtLftSen.uiRtStat));
		fUIInRtStatHide(ADR(tyP1024McSetAntiGap.tyAntiGap.tyNumLftSenOff.uiRtStat));
	ELSE
		fUIInRtStatOff(ADR(tyP1024McSetAntiGap.tyAntiGap.tyTxtLftSen.uiRtStat));
		fUIInRtStatOff(ADR(tyP1024McSetAntiGap.tyAntiGap.tyNumLftSenOff.uiRtStat));
	END_IF

	IF p_tyNtParamCurr.tyDISettings.diConvRgtSen = 0 THEN
		fUIInRtStatHide(ADR(tyP1024McSetAntiGap.tyAntiGap.tyTxtRgtSen.uiRtStat));
		fUIInRtStatHide(ADR(tyP1024McSetAntiGap.tyAntiGap.tyNumRgtSenOff.uiRtStat));
	ELSE
		fUIInRtStatOff(ADR(tyP1024McSetAntiGap.tyAntiGap.tyTxtRgtSen.uiRtStat));
		fUIInRtStatOff(ADR(tyP1024McSetAntiGap.tyAntiGap.tyNumRgtSenOff.uiRtStat));
	END_IF

	//Machine Setting - Anti Gap Sensor Filter
	tyP1024McSetAntiGap.tyAntiGap.tyNumLftSenOff.diValueMin		:= p_tyNtParamCurr.tyUIAntiGapSenOffTm.diMin;
	tyP1024McSetAntiGap.tyAntiGap.tyNumLftSenOff.diValueMax		:= p_tyNtParamCurr.tyUIAntiGapSenOffTm.diMax;

	tyP1024McSetAntiGap.tyAntiGap.tyNumRgtSenOff.diValueMin		:= p_tyNtParamCurr.tyUIAntiGapSenOffTm.diMin;
	tyP1024McSetAntiGap.tyAntiGap.tyNumRgtSenOff.diValueMax		:= p_tyNtParamCurr.tyUIAntiGapSenOffTm.diMax;

	//Parameter
	tyP1024McSetAntiGap.tyAntiGap.tyNumLftSenOff.diValue		:= p_tyMcParamCurr.tyConvLftSenAntiGapDly.diSigOffTm;

	tyP1024McSetAntiGap.tyAntiGap.tyNumRgtSenOff.diValue		:= p_tyMcParamCurr.tyConvRgtSenAntiGapDly.diSigOffTm;

END_ACTION
```

#### Act_Main_P1040.st
```iecst
(** 2018-12-21 **)
ACTION Act_Main_P1040:

//	tyP1040ProdSet.tyProdSet.tyDrpDnFlippedBrd.uiRtStat := NOT p_tyNtParamCurr.bHermesPrep;
	tyP1040ProdSet.tyProdSet.tyDrpDnFlippedBrd.uiRtStat := TRUE;
//	tyP1040ProdSet.tyProdSet.tyTxtDrpDnFlippedBrd.uiRtStat := NOT p_tyNtParamCurr.bHermesPrep;
	tyP1040ProdSet.tyProdSet.tyTxtDrpDnFlippedBrd.uiRtStat := TRUE;

	tyP1040ProdSet.tyProdSet.tyDrpDnMcMode.usiValueMinIdx	:= DINT_TO_USINT(p_tyNtParamCurr.tyProdRcpMcModLmt.diMin);
	tyP1040ProdSet.tyProdSet.tyDrpDnMcMode.usiValueMaxIdx	:= DINT_TO_USINT(p_tyNtParamCurr.tyProdRcpMcModLmt.diMax);

	tyP1040ProdSet.tyProdSet.tyNumProdWidth.diValueMin	:= p_tyNtParamCurr.tyProdRcpWidthLmt.diMin;
	tyP1040ProdSet.tyProdSet.tyNumProdWidth.diValueMax	:= p_tyNtParamCurr.tyProdRcpWidthLmt.diMax;

	tyP1040ProdSet.tyProdSet.tyDrpDnFlippedBrd.usiValueMinIdx	:= DINT_TO_USINT(p_tyNtParamCurr.tyProdRcpFlippedBrdLmt.diMin);
	tyP1040ProdSet.tyProdSet.tyDrpDnFlippedBrd.usiValueMaxIdx	:= DINT_TO_USINT(p_tyNtParamCurr.tyProdRcpFlippedBrdLmt.diMax);

	tyP1040ProdSet.tyProdSet.tyNumProdWidth2.diValueMin	:= p_tyNtParamCurr.tyProdRcpWidthLmt.diMin;
	tyP1040ProdSet.tyProdSet.tyNumProdWidth2.diValueMax	:= p_tyNtParamCurr.tyProdRcpWidthLmt.diMax;

	FOR i := 1 TO c_uiP1040TableSize DO
		tyP1040ProdSet.tyProdSet.tyTableRecipe.a_tyStringDataCol0[i].sValue	:= UINT_TO_STRING(i);
		tyP1040ProdSet.tyProdSet.tyTableRecipe.a_tyStringDataCol1[i].sValue	:= p_tyProdRcpCurrList[i].sRcpNm;
		tyP1040ProdSet.tyProdSet.tyTableRecipe.a_tyStringDataCol2[i].sValue	:= p_tyProdRcpCurrList[i].sDisplayInfo;
	END_FOR

	IF p_tyNtParamCurr.bLFProdWidth2Prep THEN
		fUIInRtStatOff(ADR(tyP1040ProdSet.tyProdSet.tyNumProdWidth2.uiRtStat));
		fUIInRtStatHide(ADR(tyP1040ProdSet.tyProdSet.tyNumProdWidth.uiRtStat));

		tyP1040ProdSet.tyProdSet.tyTableRecipe.tyStringTitle2Col2Row0.sValue:= 'US | DS Width';
	ELSE
		fUIInRtStatHide(ADR(tyP1040ProdSet.tyProdSet.tyNumProdWidth2.uiRtStat));
		fUIInRtStatOff(ADR(tyP1040ProdSet.tyProdSet.tyNumProdWidth.uiRtStat));

		tyP1040ProdSet.tyProdSet.tyTableRecipe.tyStringTitle2Col2Row0.sValue:= 'Product Width';
	END_IF

END_ACTION
```

#### Act_Main_P1050.st
```iecst
(** 2018-12-21 **)
ACTION Act_Main_P1050:

	//Leader
	//Display
	tyP1050LFSet.tyLdr.tyNumAfterOven.diValueMax	:= p_tyNtParamCurr.tyUILFIndexAfterOven.diMax;
	tyP1050LFSet.tyLdr.tyNumAfterOven.diValueMin	:= p_tyNtParamCurr.tyUILFIndexAfterOven.diMin;

	tyP1050LFSet.tyLdr.tyNumBeforeOven.diValueMax	:= p_tyNtParamCurr.tyUILFIndexBeforeOven.diMax;
	tyP1050LFSet.tyLdr.tyNumBeforeOven.diValueMin	:= p_tyNtParamCurr.tyUILFIndexBeforeOven.diMin;

	tyP1050LFSet.tyLdr.tyNumAfterOven2.diValueMax	:= p_tyNtParamCurr.tyUILFIndexAfterOven.diMax;
	tyP1050LFSet.tyLdr.tyNumAfterOven2.diValueMin	:= p_tyNtParamCurr.tyUILFIndexAfterOven.diMin;

	tyP1050LFSet.tyLdr.tyNumBeforeOven2.diValueMax	:= p_tyNtParamCurr.tyUILFIndexBeforeOven.diMax;
	tyP1050LFSet.tyLdr.tyNumBeforeOven2.diValueMin	:= p_tyNtParamCurr.tyUILFIndexBeforeOven.diMin;

	FOR i := 1 TO c_uiP1050TableSize DO
		tyP1050LFSet.tyLdr.tyTable1List.a_tyStringDataCol2[i].sValue	:= p_tyMcParamCurr.a_sLFIPAddr[i];
		tyP1050LFSet.tyLdr.tyTable1List.a_tyTxtDataCol3[i].usiValueIdx	:= (BOOL_TO_USINT(p_tyMcParamCurr.a_bLFOnline[i])) + 1;
	END_FOR

	//Parameter
	tyP1050LFSet.tyLdr.tyNumAfterOven.diValue	:= p_tyMcParamCurr.diLFMcIdxAfterOven;
	tyP1050LFSet.tyLdr.tyNumBeforeOven.diValue	:= p_tyMcParamCurr.diLFMcIdxBeforeOven;
	tyP1050LFSet.tyLdr.tyNumAfterOven2.diValue	:= p_tyMcParamCurr.diLFMcIdxAfterOven2;
	tyP1050LFSet.tyLdr.tyNumBeforeOven2.diValue	:= p_tyMcParamCurr.diLFMcIdxBeforeOven2;

END_ACTION
```

#### Act_Main_P1080.st
```iecst
(** 2018-12-21 **)
ACTION Act_Main_P1080:

	//User Managment
	FOR i := 1 TO c_uiP1080TableSize DO
		tyP1080UsrMgmt.tyUsrMgmt.tyTableList.a_tyStringDataCol0[i].sValue	:= UINT_TO_STRING(i);
		tyP1080UsrMgmt.tyUsrMgmt.tyTableList.a_tyStringDataCol1[i].sValue	:= p_tyUsrMgmtAllList[i].sUsrNm;
		tyP1080UsrMgmt.tyUsrMgmt.tyTableList.a_tyTxtDataCol3[i].usiValueIdx	:= DINT_TO_USINT((p_tyUsrMgmtAllList[i].eUsrLvl) + 1);
	END_FOR

END_ACTION
```

#### Act_Main_P1081.st
```iecst
ACTION Act_Main_P1081:

	//User Managment User Acces Right
	//Level 1
	IF p_tyUsrMgmtFullData.tyAccessRightLvl1.sNm <> '' THEN
		tyP1081UsrMgmtUsrAccessRgt.tyUsrAccessRgtLvl1.tyStringNm.sValue	:= p_tyUsrMgmtFullData.tyAccessRightLvl1.sNm;
		tyProperty.tyUITxtSnippets.sUsrMgmtUsrLv1Nm						:= p_tyUsrMgmtFullData.tyAccessRightLvl1.sNm;
	ELSE
		tyP1081UsrMgmtUsrAccessRgt.tyUsrAccessRgtLvl1.tyStringNm.sValue	:= tyProperty.tyUITxtSnippets.sUsrMgmtUsrLv1Nm;
	END_IF

	tyP1081UsrMgmtUsrAccessRgt.tyUsrAccessRgtLvl1.tyBtnOps.bValue		:= p_tyUsrMgmtFullData.tyAccessRightLvl1.bOpt;
	tyP1081UsrMgmtUsrAccessRgt.tyUsrAccessRgtLvl1.tyBtnProdSel.bValue	:= p_tyUsrMgmtFullData.tyAccessRightLvl1.bProdSel;
	tyP1081UsrMgmtUsrAccessRgt.tyUsrAccessRgtLvl1.tyBtnMagSel.bValue	:= p_tyUsrMgmtFullData.tyAccessRightLvl1.bMagSel;
	tyP1081UsrMgmtUsrAccessRgt.tyUsrAccessRgtLvl1.tyBtnMcInfo.bValue	:= p_tyUsrMgmtFullData.tyAccessRightLvl1.bMcInfo;
	tyP1081UsrMgmtUsrAccessRgt.tyUsrAccessRgtLvl1.tyBtnAlm.bValue		:= p_tyUsrMgmtFullData.tyAccessRightLvl1.bAlm;
	tyP1081UsrMgmtUsrAccessRgt.tyUsrAccessRgtLvl1.tyBtnBffrInfo.bValue	:= p_tyUsrMgmtFullData.tyAccessRightLvl1.bBffrInfo;
	tyP1081UsrMgmtUsrAccessRgt.tyUsrAccessRgtLvl1.tyBtnOvenInfo.bValue	:= p_tyUsrMgmtFullData.tyAccessRightLvl1.bOvenInfo;
	tyP1081UsrMgmtUsrAccessRgt.tyUsrAccessRgtLvl1.tyBtnMagInfo.bValue	:= p_tyUsrMgmtFullData.tyAccessRightLvl1.bMagInfo;
	tyP1081UsrMgmtUsrAccessRgt.tyUsrAccessRgtLvl1.tyBtnLFCtrl.bValue	:= p_tyUsrMgmtFullData.tyAccessRightLvl1.bLFCtrl;
	tyP1081UsrMgmtUsrAccessRgt.tyUsrAccessRgtLvl1.tyBtnManual.bValue	:= p_tyUsrMgmtFullData.tyAccessRightLvl1.bManual;
	tyP1081UsrMgmtUsrAccessRgt.tyUsrAccessRgtLvl1.tyBtnSimu.bValue		:= p_tyUsrMgmtFullData.tyAccessRightLvl1.bSimulation;
	tyP1081UsrMgmtUsrAccessRgt.tyUsrAccessRgtLvl1.tyBtnProdSet.bValue	:= p_tyUsrMgmtFullData.tyAccessRightLvl1.bProdSet;
	tyP1081UsrMgmtUsrAccessRgt.tyUsrAccessRgtLvl1.tyBtnMagSet.bValue	:= p_tyUsrMgmtFullData.tyAccessRightLvl1.bMagSet;
	tyP1081UsrMgmtUsrAccessRgt.tyUsrAccessRgtLvl1.tyBtnMcSet.bValue		:= p_tyUsrMgmtFullData.tyAccessRightLvl1.bMcSet;
	tyP1081UsrMgmtUsrAccessRgt.tyUsrAccessRgtLvl1.tyBtnLang.bValue		:= p_tyUsrMgmtFullData.tyAccessRightLvl1.bLang;
	tyP1081UsrMgmtUsrAccessRgt.tyUsrAccessRgtLvl1.tyBtnLFSet.bValue		:= p_tyUsrMgmtFullData.tyAccessRightLvl1.bLFSet;
	tyP1081UsrMgmtUsrAccessRgt.tyUsrAccessRgtLvl1.tyBtnChgParam.bValue	:= p_tyUsrMgmtFullData.tyAccessRightLvl1.bChgParam;

	//Level 2
	IF p_tyUsrMgmtFullData.tyAccessRightLvl2.sNm <> '' THEN
		tyP1081UsrMgmtUsrAccessRgt.tyUsrAccessRgtLvl2.tyStringNm.sValue	:= p_tyUsrMgmtFullData.tyAccessRightLvl2.sNm;
		tyProperty.tyUITxtSnippets.sUsrMgmtUsrLv2Nm						:= p_tyUsrMgmtFullData.tyAccessRightLvl2.sNm;
	ELSE
		tyP1081UsrMgmtUsrAccessRgt.tyUsrAccessRgtLvl2.tyStringNm.sValue	:= tyProperty.tyUITxtSnippets.sUsrMgmtUsrLv2Nm;
	END_IF

	tyP1081UsrMgmtUsrAccessRgt.tyUsrAccessRgtLvl2.tyBtnOps.bValue		:= p_tyUsrMgmtFullData.tyAccessRightLvl2.bOpt;
	tyP1081UsrMgmtUsrAccessRgt.tyUsrAccessRgtLvl2.tyBtnProdSel.bValue	:= p_tyUsrMgmtFullData.tyAccessRightLvl2.bProdSel;
	tyP1081UsrMgmtUsrAccessRgt.tyUsrAccessRgtLvl2.tyBtnMagSel.bValue	:= p_tyUsrMgmtFullData.tyAccessRightLvl2.bMagSel;
	tyP1081UsrMgmtUsrAccessRgt.tyUsrAccessRgtLvl2.tyBtnMcInfo.bValue	:= p_tyUsrMgmtFullData.tyAccessRightLvl2.bMcInfo;
	tyP1081UsrMgmtUsrAccessRgt.tyUsrAccessRgtLvl2.tyBtnAlm.bValue		:= p_tyUsrMgmtFullData.tyAccessRightLvl2.bAlm;
	tyP1081UsrMgmtUsrAccessRgt.tyUsrAccessRgtLvl2.tyBtnBffrInfo.bValue	:= p_tyUsrMgmtFullData.tyAccessRightLvl2.bBffrInfo;
	tyP1081UsrMgmtUsrAccessRgt.tyUsrAccessRgtLvl2.tyBtnOvenInfo.bValue	:= p_tyUsrMgmtFullData.tyAccessRightLvl2.bOvenInfo;
	tyP1081UsrMgmtUsrAccessRgt.tyUsrAccessRgtLvl2.tyBtnMagInfo.bValue	:= p_tyUsrMgmtFullData.tyAccessRightLvl2.bMagInfo;
	tyP1081UsrMgmtUsrAccessRgt.tyUsrAccessRgtLvl2.tyBtnLFCtrl.bValue	:= p_tyUsrMgmtFullData.tyAccessRightLvl2.bLFCtrl;
	tyP1081UsrMgmtUsrAccessRgt.tyUsrAccessRgtLvl2.tyBtnManual.bValue	:= p_tyUsrMgmtFullData.tyAccessRightLvl2.bManual;
	tyP1081UsrMgmtUsrAccessRgt.tyUsrAccessRgtLvl2.tyBtnSimu.bValue		:= p_tyUsrMgmtFullData.tyAccessRightLvl2.bSimulation;
	tyP1081UsrMgmtUsrAccessRgt.tyUsrAccessRgtLvl2.tyBtnProdSet.bValue	:= p_tyUsrMgmtFullData.tyAccessRightLvl2.bProdSet;
	tyP1081UsrMgmtUsrAccessRgt.tyUsrAccessRgtLvl2.tyBtnMagSet.bValue	:= p_tyUsrMgmtFullData.tyAccessRightLvl2.bMagSet;
	tyP1081UsrMgmtUsrAccessRgt.tyUsrAccessRgtLvl2.tyBtnMcSet.bValue		:= p_tyUsrMgmtFullData.tyAccessRightLvl2.bMcSet;
	tyP1081UsrMgmtUsrAccessRgt.tyUsrAccessRgtLvl2.tyBtnLang.bValue		:= p_tyUsrMgmtFullData.tyAccessRightLvl2.bLang;
	tyP1081UsrMgmtUsrAccessRgt.tyUsrAccessRgtLvl2.tyBtnLFSet.bValue		:= p_tyUsrMgmtFullData.tyAccessRightLvl2.bLFSet;
	tyP1081UsrMgmtUsrAccessRgt.tyUsrAccessRgtLvl2.tyBtnChgParam.bValue	:= p_tyUsrMgmtFullData.tyAccessRightLvl2.bChgParam;

	//Level 3
	IF p_tyUsrMgmtFullData.tyAccessRightLvl3.sNm <> '' THEN
		tyP1081UsrMgmtUsrAccessRgt.tyUsrAccessRgtLvl3.tyStringNm.sValue	:= p_tyUsrMgmtFullData.tyAccessRightLvl3.sNm;
		tyProperty.tyUITxtSnippets.sUsrMgmtUsrLv3Nm						:= p_tyUsrMgmtFullData.tyAccessRightLvl3.sNm;
	ELSE
		tyP1081UsrMgmtUsrAccessRgt.tyUsrAccessRgtLvl3.tyStringNm.sValue	:= tyProperty.tyUITxtSnippets.sUsrMgmtUsrLv3Nm;
	END_IF

	tyP1081UsrMgmtUsrAccessRgt.tyUsrAccessRgtLvl3.tyBtnOps.bValue		:= p_tyUsrMgmtFullData.tyAccessRightLvl3.bOpt;
	tyP1081UsrMgmtUsrAccessRgt.tyUsrAccessRgtLvl3.tyBtnProdSel.bValue	:= p_tyUsrMgmtFullData.tyAccessRightLvl3.bProdSel;
	tyP1081UsrMgmtUsrAccessRgt.tyUsrAccessRgtLvl3.tyBtnMagSel.bValue	:= p_tyUsrMgmtFullData.tyAccessRightLvl3.bMagSel;
	tyP1081UsrMgmtUsrAccessRgt.tyUsrAccessRgtLvl3.tyBtnMcInfo.bValue	:= p_tyUsrMgmtFullData.tyAccessRightLvl3.bMcInfo;
	tyP1081UsrMgmtUsrAccessRgt.tyUsrAccessRgtLvl3.tyBtnAlm.bValue		:= p_tyUsrMgmtFullData.tyAccessRightLvl3.bAlm;
	tyP1081UsrMgmtUsrAccessRgt.tyUsrAccessRgtLvl3.tyBtnBffrInfo.bValue	:= p_tyUsrMgmtFullData.tyAccessRightLvl3.bBffrInfo;
	tyP1081UsrMgmtUsrAccessRgt.tyUsrAccessRgtLvl3.tyBtnOvenInfo.bValue	:= p_tyUsrMgmtFullData.tyAccessRightLvl3.bOvenInfo;
	tyP1081UsrMgmtUsrAccessRgt.tyUsrAccessRgtLvl3.tyBtnMagInfo.bValue	:= p_tyUsrMgmtFullData.tyAccessRightLvl3.bMagInfo;
	tyP1081UsrMgmtUsrAccessRgt.tyUsrAccessRgtLvl3.tyBtnLFCtrl.bValue	:= p_tyUsrMgmtFullData.tyAccessRightLvl3.bLFCtrl;
	tyP1081UsrMgmtUsrAccessRgt.tyUsrAccessRgtLvl3.tyBtnManual.bValue	:= p_tyUsrMgmtFullData.tyAccessRightLvl3.bManual;
	tyP1081UsrMgmtUsrAccessRgt.tyUsrAccessRgtLvl3.tyBtnSimu.bValue		:= p_tyUsrMgmtFullData.tyAccessRightLvl3.bSimulation;
	tyP1081UsrMgmtUsrAccessRgt.tyUsrAccessRgtLvl3.tyBtnProdSet.bValue	:= p_tyUsrMgmtFullData.tyAccessRightLvl3.bProdSet;
	tyP1081UsrMgmtUsrAccessRgt.tyUsrAccessRgtLvl3.tyBtnMagSet.bValue	:= p_tyUsrMgmtFullData.tyAccessRightLvl3.bMagSet;
	tyP1081UsrMgmtUsrAccessRgt.tyUsrAccessRgtLvl3.tyBtnMcSet.bValue		:= p_tyUsrMgmtFullData.tyAccessRightLvl3.bMcSet;
	tyP1081UsrMgmtUsrAccessRgt.tyUsrAccessRgtLvl3.tyBtnLang.bValue		:= p_tyUsrMgmtFullData.tyAccessRightLvl3.bLang;
	tyP1081UsrMgmtUsrAccessRgt.tyUsrAccessRgtLvl3.tyBtnLFSet.bValue		:= p_tyUsrMgmtFullData.tyAccessRightLvl3.bLFSet;
	tyP1081UsrMgmtUsrAccessRgt.tyUsrAccessRgtLvl3.tyBtnChgParam.bValue	:= p_tyUsrMgmtFullData.tyAccessRightLvl3.bChgParam;

END_ACTION
```

#### Act_Background.st - Do Not Change!!!
```iecst
(** 2018-12-10 **)
ACTION Act_Background:

	//Main
	Act_ChgPage;
	Act_OptPage;

END_ACTION
```

#### Package Logical/UI/UI/Act_Background - Change By Project

#### Act_ChgPage.st
```iecst
(** 2020-10-08 **)
ACTION Act_ChgPage:

	(*Exit Page*)
	IF (eChgPage <> eChgPageOld) OR (usiChgPage = 2) AND p_bStartupRun = FALSE THEN

		usiChgPage	:= 2;

		CASE eChgPageOld OF
			UIP0700LFCtrl:
				Act_ExitP0700;

			UIP1000Lang:
				Act_ExitP1000;

			UIP1021McSetGen:
				Act_ExitP1021;

			UIP1022McSetVComm:
				Act_ExitP1022;

			UIP1023McSetHComm:
				Act_ExitP1023;

			UIP1024McSetAntiGap:
				Act_ExitP1024;

			UIP1080UsrMgmt:
				Act_ExitP1080;

			UIP1081UsrMgmtUsrAccessRgt:
				Act_ExitP1081;

			ELSE
				usiChgPage	:= 1;

		END_CASE

		IF usiChgPage = 1 THEN
			eChgPageOld		:= eChgPage;
		END_IF

	(*Enter Page*)
	ELSIF usiChgPage = 1 THEN

		CASE eChgPage OF

			UIP0001Startup:
				Act_EntP0001Disp;

			UIP0002Menu:
				Act_EntP0002Disp;

			UIP0100Login:
				Act_EntP0100Disp;

			UIP0200OpsGen:
				Act_EntP0200Disp;

			UIP0201OpsConv:
				Act_EntP0201Disp;

			UIP0300McInfo:
				Act_EntP0300Disp;

			UIP0400ProdSel:
				Act_EntP0400Disp;

			UIP0600Alm:
				Act_EntP0600Disp;

			UIP0700LFCtrl:
				Act_EntP0700Disp;

			UIP0900GenIn:
				Act_EntP0900Disp;

			UIP0910GenOut:
				Act_EntP0910Disp;

			UIP0920MtrNPneuCtrl:
				Act_EntP0920Disp;

			UIP0921ClampNoRS:
				Act_EntP0921Disp;

			UIP0922Shutter:
				Act_EntP0922Disp;

			UIP0923Stopper:
				Act_EntP0923Disp;

			UIP0924ClampWithRS:
				Act_EntP0924Disp;

			UIP0931ConvInv:
				Act_EntP0931Disp;

			UIP0934AW:
				Act_EntP0934Disp;

			UIP0940CommCtrl:
				Act_EntP0940Disp;

			UIP0950Simu:
				Act_EntP0950Disp;

			UIP1000Lang:
				Act_EntP1000Disp;

			UIP1020McSetNavi:
				Act_EntP1020Disp;

			UIP1021McSetGen:
				Act_EntP1021Disp;

			UIP1022McSetVComm:
				Act_EntP1022Disp;

			UIP1023McSetHComm:
				Act_EntP1023Disp;

			UIP1024McSetAntiGap:
				Act_EntP1024Disp;

			UIP1040ProdSet:
				Act_EntP1040Disp;

			UIP1050LFSet:
				Act_EntP1050Disp;

			UIP1080UsrMgmt:
				Act_EntP1080Disp;

			UIP1081UsrMgmtUsrAccessRgt:
				Act_EntP1081Disp;

		END_CASE

		usiChgPage	:= 0;

		tyProperty.tyVisu.uiChgPage	:= UDINT_TO_UINT(eChgPage);

	END_IF

END_ACTION
```

#### Act_OptPage.st
```iecst
(** 2020-10-08 **)
ACTION Act_OptPage:

	//Prevent Screen Saver Interupt Program
	IF tyProperty.tyVisu.uiCurrPage <> 0 THEN
		eCurrPage := tyProperty.tyVisu.uiCurrPage;
	ELSE
		Act_OptP0000McStatus;
		Act_OptP0000RunningNm;
		Act_OptP0000StatDisp;
	END_IF

	Act_OptP0000DisableSSaver;
	Act_OptP0000TouchTimer;

	Act_OptP0002ToP1081UnlockCoverPB;

	IF (tyProperty.tyVisu.uiChgPage = 65535) AND (usiChgPage = 0) THEN

		Act_OptC0005GoHomeCtrl;
		Act_OptC0005ShowNotif;
		Act_OptC0005AutoCtrl;
		Act_OptC0005RstErr;
		Act_OptC0005StatBarCtrl;
		Act_OptC0005Buzzer;
		Act_OptC0005ChgPage;
		Act_OptC0007Notif;
		Act_OptC0009Info;
		Act_OptC0011Loading;

		CASE eCurrPage OF
			UIP0001Startup:
				Act_OptP0001Startup;

			UIP0100Login:
				Act_OptP0100Keypad;
				Act_OptP0100NomLogin;
				Act_OptP0100BypassLogin;
				Act_OptP0100Logout;

			UIP0200OpsGen:
				Act_OptP0200ChgPage;
				Act_OptP0200UpdtDat;
				Act_OptP0200VSMEMA;
				Act_OptP0200RcyMsg;
				Act_OptP0200ToP0201AccDat;
				Act_OptP0200ToP0201BypsInitConv;
				Act_OptP0200ToP0201RlsNewProd;
				Act_OptP0200PCBReset;

			UIP0201OpsConv:
				Act_OptP0201Navi;
				Act_OptP0201UpdtDat;
				Act_OptP0201IOMonitor;
				Act_OptP0201ChgParam;
				Act_OptP0201Keypad;
				Act_OptP0200ToP0201AccDat;
				Act_OptP0200ToP0201BypsInitConv;
				Act_OptP0200ToP0201RlsNewProd;

			UIP0300McInfo:
				Act_OptP0300Song;

			UIP0400ProdSel:
				Act_OptP0400Search;
				Act_OptP0400Load;
				Act_OptP0400Preview;
				Act_OptP0400Table;
				Act_OptP0400Keypad;
				Act_OptP0400Mask;
				Act_OptP0400Sort;
				Act_OptP0400RcpPopUp;

			UIP0600Alm:
				Act_OptP0600Alm;
				Act_OptP0600RcyMsg;

			UIP0700LFCtrl:
				Act_OptP0700LFLeaderCtrl;
				Act_OptP0700Mask;
				Act_OptP0700Table;

			UIP0002Menu, UIP0900GenIn, UIP0910GenOut, UIP0920MtrNPneuCtrl,UIP0921ClampNoRS, UIP0922Shutter, UIP0923Stopper, UIP0924ClampWithRS, UIP0931ConvInv, UIP0934AW, UIP0940CommCtrl:
				IF eCurrPage = UIP0002Menu THEN
					Act_OptP0002ChgPage;
					Act_OptP0002Mask;
					Act_OptP0002UpdtData;
					Act_OptP0002PCBReset;
				END_IF

				Act_OptP0002ManualCtrl;
				Act_OptP0910RstMnl;
				Act_OptP0921RstMnl;
				Act_OptP0922RstMnl;
				Act_OptP0923RstMnl;
				Act_OptP0924RstMnl;
				Act_OptP0931RstMnl;
				Act_OptP0934RstMnl;
				Act_OptP0940RstMnl;

				IF bUIManualMod THEN
					//General Input
					Act_OptP0900ReadDI;

					//General Output
					Act_OptP0910WriteDO;

					//MtrNPneuCtrl
					Act_OptP0920FullMask;
					Act_OptP0920ChgPage;

					//Clamp No RS Ctrl
					Act_OptP0921FullMask;
					Act_OptP0921Navi;
					Act_OptP0921ChgLyr;
					Act_OptP0921UpdtData;
					Act_OptP0921FBCtrl;
					Act_OptP0921FBStat;
					Act_OptP0921DCCtrl;

					//Inlet & Outlet Shutter
					Act_OptP0922DualMask;
					Act_OptP0922Navi;
					Act_OptP0922InletShutterChgLyr;
					Act_OptP0922InletShutterSen;
					Act_OptP0922InletShutterFB;
					Act_OptP0922InletShutterFBStat;
					Act_OptP0922InletShutterDC;
					Act_OptP0922OutletShutterChgLyr;
					Act_OptP0922OutletShutterSen;
					Act_OptP0922OutletShutterFB;
					Act_OptP0922OutletShutterFBStat;
					Act_OptP0922OutletShutterDC;

					//Stopper Ctrl
					Act_OptP0923FullMask;
					Act_OptP0923Navi;
					Act_OptP0923ChgLyr;
					Act_OptP0923UpdtData;
					Act_OptP0923FBCtrl;
					Act_OptP0923FBStat;
					Act_OptP0923DCCtrl;

					//Clamp With RS 1&2&3
					Act_OptP0924DualMask;
					Act_OptP0924Navi;
					Act_OptP0924Clamp1ChgLyr;
					Act_OptP0924Clamp1Sen;
					Act_OptP0924Clamp1FB;
					Act_OptP0924Clamp1FBStat;
					Act_OptP0924Clamp1DC;

					Act_OptP0924Clamp2ChgLyr;
					Act_OptP0924Clamp2Sen;
					Act_OptP0924Clamp2FB;
					Act_OptP0924Clamp2FBStat;
					Act_OptP0924Clamp2DC;

					Act_OptP0924Clamp3ChgLyr;
					Act_OptP0924Clamp3Sen;
					Act_OptP0924Clamp3FB;
					Act_OptP0924Clamp3FBStat;
					Act_OptP0924Clamp3DC;

					//Conveyor and Inverter
					Act_OptP0931DualMask;
					Act_OptP0931Navi;
					Act_OptP0931Sen;
					Act_OptP0931ConvChgLyr;
					Act_OptP0931ConvFB;
					Act_OptP0931ConvFBStat;
					Act_OptP0931ConvDC;
					Act_OptP0931InvChgLyr;
					Act_OptP0931InvUpdtData;
					Act_OptP0931InvFB;
					Act_OptP0931InvFBStat;
					Act_OptP0931InvDC;

					//AutoWidth
					Act_OptP0934FullMask;
					Act_OptP0934Navi;
					Act_OptP0934FB;
					Act_OptP0934FBStat;
					Act_OptP0934Mask;
					Act_OptP0934UpdtDat;
					Act_OptP0934Keypad;

					//Communication
					Act_OptP0940FullMask;
					Act_OptP0940ReadDI;
					Act_OptP0940WriteDO;

				END_IF

			UIP0950Simu:
				Act_OptP0950Control;
				Act_OptP0950SimulationMod;

			UIP1000Lang:
				Act_OptP1000SelectLang;
				Act_OptP1000Keypad;

			UIP1020McSetNavi:
				Act_OptP1020Navi;

			UIP1021McSetGen:
				Act_OptP1021Navi;
				Act_OptP1021Save;
				Act_OptP1021Keypad;
				Act_OptP1021IPAddr;
				Act_OptP1021SubnetMask;
				Act_OptP1021DHCPSetting;

			UIP1022McSetVComm:
				Act_OptP1022Navi;
				Act_OptP1022Save;
				Act_OptP1022DisLF;

			UIP1023McSetHComm:
				Act_OptP1023Navi;
				Act_OptP1023ShowLyr;
				Act_OptP1023Save;
				Act_OptP1023USSel;
				Act_OptP1023DSSel;
				Act_OptP1023Keypad;

			UIP1024McSetAntiGap:
				Act_OptP1024Navi;
				Act_OptP1024Save;
				Act_OptP1024Keypad;

			UIP1040ProdSet:
				Act_OptP1040Mask;
				Act_OptP1040Save;
				Act_OptP1040Del;
				Act_OptP1040Table;
				Act_OptP1040LoadData;
				Act_OptP1040Search;
				Act_OptP1040Keypad;
				Act_OptP1040ToXML;
				Act_OptP1040FromXML;
				Act_OptP1040Sort;
				Act_OptP1040RcpPopUp;

			UIP1050LFSet:
				Act_OptP1050Keypad;
				Act_OptP1050Edit;
				Act_OptP1050Online;
				Act_OptP1050Offline;
				Act_OptP1050Delete;
				Act_OptP1050ShftUp;
				Act_OptP1050ShftDwn;
				Act_OptP1050Mask;
				Act_OptP1050Table;

			UIP1080UsrMgmt:
				Act_OptP1080AddUsr;
				Act_OptP1080DelUsr;
				Act_OptP1080EditUsr;
				Act_OptP1080EditAccess;
				Act_OptP1080Table;
				Act_OptP1080Keypad;

			UIP1081UsrMgmtUsrAccessRgt:
				Act_OptP1081Navi;
				Act_OptP1081Load;
				Act_OptP1081Save;
				Act_OptP1081Keypad;

		END_CASE

	END_IF

END_ACTION
```

#### Act_OptC0004NaviP1024.st
```iecst
ACTION Act_OptC0004NaviP1024:

	IF tyP1024McSetAntiGap.tyNaviBack.tyBtnBack.bRtCompl = TRUE THEN
		IF usiSaveMcParamStep = 255 THEN
			eChgPage			:= eCurrPage;
			usiSaveMcParamStep	:= 0;

			tyP1024McSetAntiGap.tyNaviBack.tyBtnBack.bRtCompl	:= FALSE;

		ELSIF usiSaveMcParamStep = 99 THEN
			usiSaveMcParamStep	:= 0;
			eChgPage			:= UIP1020McSetNavi;

			Act_ExitC0006RstBtn;

			tyP1024McSetAntiGap.tyNaviBack.tyBtnBack.bRtCompl	:= FALSE;

		ELSE
			Act_ExitP1024Save;

		END_IF
	END_IF

END_ACTION
```

#### Act_OptC0005GoHomeCtrl.st
```iecst
ACTION Act_OptC0005GoHomeCtrl:

	//Control
	IF tyCommon.tyMain.tyBtnHome.bRtCompl = TRUE THEN
		tyCommon.tyMain.tyBtnHome.bRtCompl	:= FALSE;

		eChgPage	:= UIP0002Menu;
	END_IF

	//Mask
	IF tyP0100Login.tyLogin.tyBtnLogin.bRtCompl 				OR tyP0100Login.tyLogout.tyBtnLogout.bRtCompl
		OR tyP0400ProdSel.tyProdSel.tyBtnLoad.bRtCompl 			OR tyP0400ProdSel.tyProdSel.tyStringSearch.bRtCompl
		OR tyP1040ProdSet.tyProdSet.tyBtnToXML.bRtCompl 		OR tyP1040ProdSet.tyProdSet.tyBtnFromXML.bRtCompl
		OR tyP1040ProdSet.tyProdSet.tyBtnDelete.bRtCompl 		OR tyP1040ProdSet.tyProdSet.tyBtnSave.bRtCompl
		OR tyP1050LFSet.tyLdr.tyBtnDelete.bRtCompl 				OR tyP1050LFSet.tyLdr.tyBtnOnline.bRtCompl
		OR tyP1050LFSet.tyLdr.tyBtnOffline.bRtCompl				OR tyP1050LFSet.tyLdr.tyBtnShftUp.bRtCompl
		OR tyP1050LFSet.tyLdr.tyBtnShftDwn.bRtCompl				OR tyP1080UsrMgmt.tyUsrMgmt.tyBtnDeleteUsr.bRtCompl
		OR tyP1080UsrMgmt.tyUsrMgmt.tyBtnEditDetail.bRtCompl	OR tyP1080UsrMgmt.tyUsrMgmt.tyBtnNewUsr.bRtCompl
		OR tyCommon.tySet.tyBtnSave.bRtCompl THEN

		fUIInRtStatOff(ADR(tyCommon.tyMain.tyBtnHome.uiMaskRtStat));

	ELSIF bUIManualMod THEN
		fUIInRtStatHide(ADR(tyCommon.tyMain.tyBtnHome.uiMaskRtStat));

	ELSE
		fUIInRtStatHide(ADR(tyCommon.tyMain.tyBtnHome.uiMaskRtStat));

	END_IF

END_ACTION
```

#### Act_OptC0005ShowNotif.st
```iecst
ACTION Act_OptC0005ShowNotif:

	//Control
	IF tyCommon.tyMain.tyBtnNotification.bRtCompl = TRUE THEN
		tyCommon.tyMain.tyBtnNotification.bRtCompl	:= FALSE;

		fUIInRtStatOff(ADR(tyCommon.tyNotif.tyLyr.uiRtStat));
	END_IF

END_ACTION
```

#### Act_OptC0005RstErr.st
```iecst
ACTION Act_OptC0005RstErr:

	//Control
	IF tyCommon.tyMain.tyBtnReset.bRtCompl = TRUE THEN
		eRstErrAct	:= RstErrActRun;

		IF p_eRstErrStat = RstErrActRun AND p_eRstErrStatus =  Done THEN
			eRstErrAct	:= RstErrActIdle;

			IF p_tyNtParamCurr.bProjCoatingPrep THEN
				bLoadingScreen:= TRUE;
			END_IF

			tyCommon.tyMain.tyBtnReset.bRtCompl	:= FALSE;
		END_IF

	END_IF

	//Mask
	IF p_bAlarmErr = TRUE OR p_bAlarmWarning = TRUE OR p_bAlarmInfo = TRUE OR p_tyDI.bSafetyRlySig = FALSE THEN
		fUIInRtStatHide(ADR(tyCommon.tyMain.tyBtnReset.uiMaskRtStat));
		bLoadingScreen:= FALSE;
	ELSE
		fUIInRtStatOff(ADR(tyCommon.tyMain.tyBtnReset.uiMaskRtStat));
	END_IF

END_ACTION
```

#### Act_OptC0005StatBarCtrl.st
```iecst
ACTION Act_OptC0005StatBarCtrl:

	//Error / Warning / Info
	IF p_bAlarmErr = TRUE OR p_bAlarmWarning = TRUE OR p_bAlarmInfo = TRUE THEN

		fbErrBlinkTm(IN := TRUE);
		IF fbErrBlinkTm.Q = TRUE THEN
			fbErrBlinkTm(IN := FALSE);

			IF p_bAlarmErr = TRUE THEN

				IF tyCommon.tyMain.tyBitmapStatBar.usiValueIdx = 1 THEN
					tyCommon.tyMain.tyBitmapStatBar.usiValueIdx	:= 0;
				ELSE
					tyCommon.tyMain.tyBitmapStatBar.usiValueIdx	:= 1;
				END_IF

			ELSE

				IF tyCommon.tyMain.tyBitmapStatBar.usiValueIdx = 3 THEN
					tyCommon.tyMain.tyBitmapStatBar.usiValueIdx	:= 0;
				ELSE
					tyCommon.tyMain.tyBitmapStatBar.usiValueIdx	:= 3;
				END_IF

			END_IF

		END_IF

	//Safety Relay Signal Activated
	ELSIF p_tyDI.bSafetyRlySig = FALSE THEN

		fbRstBlinkTm(IN := TRUE);
		IF fbRstBlinkTm.Q = TRUE THEN
			fbRstBlinkTm(IN := FALSE);

			IF tyCommon.tyMain.tyBitmapStatBar.usiValueIdx = 5 THEN
				tyCommon.tyMain.tyBitmapStatBar.usiValueIdx	:= 6;
			ELSE
				tyCommon.tyMain.tyBitmapStatBar.usiValueIdx	:= 5;
			END_IF

		END_IF

	//Manual Running
	ELSIF bUIManualMod THEN
		tyCommon.tyMain.tyBitmapStatBar.usiValueIdx	:= 7;

	//Operation Cycle Stopping
	ELSIF p_eOpsOpsStatus = OperationsStatusCycleStopping THEN

		fbStopBlinkTm(IN := TRUE);
		IF fbStopBlinkTm.Q = TRUE THEN
			fbStopBlinkTm(IN := FALSE);

			IF tyCommon.tyMain.tyBitmapStatBar.usiValueIdx = 1 THEN
				tyCommon.tyMain.tyBitmapStatBar.usiValueIdx	:= 2;
			ELSE
				tyCommon.tyMain.tyBitmapStatBar.usiValueIdx	:= 1;
			END_IF

		END_IF

	//Operation Stepping
	ELSIF p_eOpsOpsStatus = OperationsStatusStep THEN
		tyCommon.tyMain.tyBitmapStatBar.usiValueIdx	:= 3;

	//Operation Running
	ELSIF p_eOpsOpsStatus = OperationsStatusRun THEN
		tyCommon.tyMain.tyBitmapStatBar.usiValueIdx	:= 2;

	//Standby
	ELSE
		tyCommon.tyMain.tyBitmapStatBar.usiValueIdx	:= 0;

	END_IF

END_ACTION
```

#### Act_OptC0005AutoCtrl.st
```iecst
ACTION Act_OptC0005AutoCtrl:

	//Control
	//Error
	IF EDGEPOS(p_bAlarmErr = TRUE AND p_bOpsStatusStop = FALSE) THEN

		tyCommon.tyMain.tyBtnStart.bRtCompl	:= FALSE;
		tyCommon.tyMain.tyBtnStop.bRtCompl	:= FALSE;
		tyCommon.tyMain.tyBtnStep.bRtCompl	:= FALSE;

		tyCommon.tyMain.tyBtnStart.bValue	:= FALSE;
		tyCommon.tyMain.tyBtnStop.bValue	:= FALSE;
		tyCommon.tyMain.tyBtnStep.bValue	:= FALSE;

		eOpsAct	:= OperationsActError;

	ELSE

		IF p_eOpsStat = OperationsActError AND p_eOpsStatus = Done THEN
			eOpsAct	:= OperationsActIdle;
		END_IF

	END_IF

	//Start
	IF tyCommon.tyMain.tyBtnStart.bRtCompl = TRUE THEN

		IF tyCommon.tyMain.tyBtnStart.bValue = TRUE THEN

			IF eCurrPage <> UIP0200OpsGen AND eCurrPage <> UIP0201OpsConv THEN

				IF bChgPage = FALSE THEN
					bChgPage	:= TRUE;
					eChgPage	:= UIP0200OpsGen;
				ELSE
					IF eChgPage <> UIP0200OpsGen THEN
						bChgPage	:= FALSE;

						tyCommon.tyMain.tyBtnStart.bRtCompl	:= FALSE;
						tyCommon.tyMain.tyBtnStart.bValue	:= FALSE;
					END_IF
				END_IF

			ELSE
				bChgPage	:= FALSE;

				tyCommon.tyMain.tyBtnStart.bValue	:= FALSE;

				tyCommon.tyMain.tyBtnStop.bRtCompl	:= FALSE;
				tyCommon.tyMain.tyBtnStep.bRtCompl	:= FALSE;

				tyCommon.tyMain.tyBtnStop.bValue	:= FALSE;
				tyCommon.tyMain.tyBtnStep.bValue	:= FALSE;
			END_IF

		ELSE

			eOpsAct	:= OperationsActStart;

			IF p_eOpsStat = OperationsActStart AND p_eOpsStatus = Done THEN
				eOpsAct	:= OperationsActIdle;

				tyCommon.tyMain.tyBtnStart.bRtCompl	:= FALSE;
			END_IF

		END_IF

	END_IF

	//Stop
	IF tyCommon.tyMain.tyBtnStop.bRtCompl = TRUE THEN

		IF tyCommon.tyMain.tyBtnStop.bValue = TRUE THEN

			tyCommon.tyMain.tyBtnStop.bValue	:= FALSE;

			tyCommon.tyMain.tyBtnStart.bRtCompl	:= FALSE;
			tyCommon.tyMain.tyBtnStep.bRtCompl	:= FALSE;

			tyCommon.tyMain.tyBtnStart.bValue	:= FALSE;
			tyCommon.tyMain.tyBtnStep.bValue	:= FALSE;

		ELSE

			eOpsAct	:= OperationsActStop;

			IF p_eOpsStat = OperationsActStop AND p_eOpsStatus = Done THEN
				eOpsAct	:= OperationsActIdle;

				tyCommon.tyMain.tyBtnStop.bRtCompl	:= FALSE;
			END_IF

		END_IF

	END_IF

	//Step
	IF tyCommon.tyMain.tyBtnStep.bRtCompl = TRUE THEN

		IF tyCommon.tyMain.tyBtnStep.bValue = TRUE THEN

			IF eCurrPage <> UIP0200OpsGen AND eCurrPage <> UIP0201OpsConv THEN

				IF bChgPage = FALSE THEN
					bChgPage	:= TRUE;
					eChgPage	:= UIP0200OpsGen;
				ELSE
					IF eChgPage <> UIP0200OpsGen THEN
						bChgPage	:= FALSE;

						tyCommon.tyMain.tyBtnStep.bRtCompl	:= FALSE;
						tyCommon.tyMain.tyBtnStep.bValue	:= FALSE;
					END_IF
				END_IF

			ELSE
				bChgPage	:= FALSE;

				tyCommon.tyMain.tyBtnStep.bValue	:= FALSE;

				tyCommon.tyMain.tyBtnStart.bRtCompl	:= FALSE;
				tyCommon.tyMain.tyBtnStop.bRtCompl	:= FALSE;

				tyCommon.tyMain.tyBtnStart.bValue	:= FALSE;
				tyCommon.tyMain.tyBtnStop.bValue	:= FALSE;
			END_IF

		ELSE

			eOpsAct	:= OperationsActStep;

			IF p_eOpsStat = OperationsActStep AND p_eOpsStatus = Done THEN
				eOpsAct	:= OperationsActIdle;

				tyCommon.tyMain.tyBtnStep.bRtCompl	:= FALSE;
			END_IF

		END_IF

	END_IF

	//Display
	//Auto Step
	IF p_tyMcParamCurr.bAutoStepEn = TRUE THEN
		fUIInRtStatOff(ADR(tyCommon.tyMain.tyBtnStep.uiRtStat));
	ELSE
		fUIInRtStatHide(ADR(tyCommon.tyMain.tyBtnStep.uiRtStat));
		fUIInRtStatHide(ADR(tyCommon.tyMain.tyBtnStep.uiMaskRtStat));
	END_IF

	//Mask
	IF (p_bAlarmErr = TRUE) OR (bUIManualMod = TRUE) OR (p_tyDI.bSafetyRlySig = FALSE) OR (tyCommon.tyMain.tyBtnHome.uiMaskRtStat.0 = FALSE) OR (bBypassTopCover1 AND NOT(p_bOpsRun)) THEN
		fUIInRtStatOff(ADR(tyCommon.tyMain.tyBtnStart.uiMaskRtStat));
		fUIInRtStatOff(ADR(tyCommon.tyMain.tyBtnStop.uiMaskRtStat));

		IF p_tyMcParamCurr.bAutoStepEn = TRUE THEN
			fUIInRtStatOff(ADR(tyCommon.tyMain.tyBtnStep.uiMaskRtStat));
		END_IF

	ELSE

		IF p_bOpsStatusRun = TRUE THEN

			fUIInRtStatOff(ADR(tyCommon.tyMain.tyBtnStart.uiMaskRtStat));
			fUIInRtStatHide(ADR(tyCommon.tyMain.tyBtnStop.uiMaskRtStat));
			fUIInRtStatHide(ADR(tyCommon.tyMain.tyBtnStep.uiMaskRtStat));

		ELSIF p_bOpsStatusCycleStop = TRUE THEN

			fUIInRtStatHide(ADR(tyCommon.tyMain.tyBtnStart.uiMaskRtStat));
			fUIInRtStatOff(ADR(tyCommon.tyMain.tyBtnStop.uiMaskRtStat));
			fUIInRtStatHide(ADR(tyCommon.tyMain.tyBtnStep.uiMaskRtStat));

		ELSIF p_bOpsStatusStep = TRUE THEN

			fUIInRtStatHide(ADR(tyCommon.tyMain.tyBtnStart.uiMaskRtStat));
			fUIInRtStatHide(ADR(tyCommon.tyMain.tyBtnStop.uiMaskRtStat));

			IF p_eOpsStatus = Busy THEN
				fUIInRtStatOff(ADR(tyCommon.tyMain.tyBtnStep.uiMaskRtStat));
			ELSE
				fUIInRtStatHide(ADR(tyCommon.tyMain.tyBtnStep.uiMaskRtStat));
			END_IF

		ELSE

			IF bDSTranErr = TRUE THEN
				fUIInRtStatOff(ADR(tyCommon.tyMain.tyBtnStart.uiMaskRtStat));
			ELSE
				fUIInRtStatHide(ADR(tyCommon.tyMain.tyBtnStart.uiMaskRtStat));
			END_IF

			fUIInRtStatOff(ADR(tyCommon.tyMain.tyBtnStop.uiMaskRtStat));
			fUIInRtStatHide(ADR(tyCommon.tyMain.tyBtnStep.uiMaskRtStat));

		END_IF

	END_IF

	IF p_bDSSMEMAAlmData.udiCode = 10000  OR p_bConvAlmData.udiCode=10114 OR p_bConvAlmData.udiCode=10119 THEN
		bDSTranErr := TRUE;
	END_IF

	IF p_tyDI.bConvRgtSen = FALSE AND p_tyDI.bConvLftSen = FALSE  THEN
		bDSTranErr := FALSE;
	END_IF

END_ACTION
```

#### Act_OptC0005Buzzer.st
```iecst
ACTION Act_OptC0005Buzzer:

	IF tyCommon.tyMain.tyBtnMuteBuz.bRtCompl = TRUE THEN
		tyCommon.tyMain.tyBtnMuteBuz.bRtCompl	:= FALSE;

		IF tyCommon.tyMain.tyBtnMuteBuz.bValue = TRUE THEN
			tyCommon.tyMain.tyBtnMuteBuz.usiBitmapIdx	:= 2;

			bMuteBuz	:= TRUE;
		ELSE
			tyCommon.tyMain.tyBtnMuteBuz.usiBitmapIdx	:= 1;

			bMuteBuz	:= FALSE;
		END_IF

	END_IF

	//Mute Buzzer
	IF EDGEPOS(p_bAlarmErr OR p_bAlarmWarning OR p_bAlarmInfo) (*AND NOT bUIManualMod)*) THEN
		tyCommon.tyMain.tyBtnMuteBuz.bValue				:= FALSE;
		tyCommon.tyMain.tyBtnMuteBuz.bRtLk				:= FALSE;
		tyCommon.tyMain.tyBtnMuteBuz.usiBitmapIdx		:= 1;

		bMuteBuz	:= FALSE;

	ELSIF NOT(p_bAlarmErr OR p_bAlarmWarning OR p_bAlarmInfo) (*OR bUIManualMod*) THEN
		tyCommon.tyMain.tyBtnMuteBuz.bRtLk				:= TRUE;
		tyCommon.tyMain.tyBtnMuteBuz.usiBitmapIdx		:= 0;

		bMuteBuz	:= FALSE;
	END_IF

END_ACTION
```

#### Act_OptC0005ChgPage.st
```iecst
ACTION Act_OptC0005ChgPage:

	IF tyCommon.tyMain.tyHotspotNaviStart.bRtCompl = TRUE THEN
		tyCommon.tyMain.tyHotspotNaviStart.bRtCompl := FALSE;

		IF p_bAlarmErr = TRUE OR p_bAlarmWarning THEN
			eChgPage 	:=UIP0600Alm;
		END_IF

	END_IF

	//Display Alarm Button Control
	tyCommon.tyMain.tyHotspotNaviStart.uiRtStat.0	:=tyCommon.tyMain.tyBtnStart.uiMaskRtStat.0;

END_ACTION
```

#### Act_OptC0007Notif.st
```iecst
ACTION Act_OptC0007Notif:

	//Display
	//User Level
	tyCommon.tyNotif.tyStringUsrNm.sValue	:= p_tyUsrMgmtCurrUsr.sUsrNm;
	tyCommon.tyNotif.tyTxtUsrLv.usiValueIdx	:= UDINT_TO_USINT(p_tyUsrMgmtCurrUsr.eUsrLvl);
	tyCommon.tyNotif.tyTxtLFMc.uiRtStat.0	:= NOT (p_tyNtParamCurr.bLFPrep AND p_tyMcParamCurr.bLFEn);

	IF p_tyNtParamCurr.bLFUsrSetPrep = TRUE THEN
		IF p_tyMcParamCurr.bLFLeaderMc = TRUE THEN
			tyCommon.tyNotif.tyTxtLFMc.usiValueIdx		:= 0;
		ELSE
			IF p_tyMcParamCurr.bSectionLeader = TRUE THEN
				tyCommon.tyNotif.tyTxtLFMc.usiValueIdx		:= 2;
			ELSE
				tyCommon.tyNotif.tyTxtLFMc.usiValueIdx		:= 1;
			END_IF
		END_IF
	END_IF

	//Info
	tyCommon.tyNotif.tyBitmapShowInfo.uiRtStat.0	:= p_bAlarmInfo = FALSE;
	tyCommon.tyNotif.tyHotspotShowInfo.uiRtStat.0	:= p_bAlarmInfo = FALSE;

	//Control
	IF tyCommon.tyNotif.tyLyr.uiRtStat.0 = FALSE THEN

		IF tyCommon.tyNotif.tyHotspotClose.bRtCompl = TRUE THEN
			tyCommon.tyNotif.tyHotspotClose.bRtCompl	:= FALSE;

			fUIInRtStatHide(ADR(tyCommon.tyNotif.tyLyr.uiRtStat));

		ELSIF tyCommon.tyNotif.tyHotspotShowInfo.bRtCompl = TRUE THEN
			tyCommon.tyNotif.tyHotspotShowInfo.bRtCompl	:= FALSE;

			fUIInRtStatOff(ADR(tyCommon.tyInfo.tyLyr.uiRtStat));
			fUIInRtStatHide(ADR(tyCommon.tyNotif.tyLyr.uiRtStat));

		END_IF

	END_IF

END_ACTION
```

#### Act_OptC0009Info.st
```iecst
ACTION Act_OptC0009Info:

	//Display
	IF EDGEPOS(p_bAlarmInfo) THEN
		fUIInRtStatOff(ADR(tyCommon.tyInfo.tyLyr.uiRtStat));

	ELSIF EDGENEG(p_bAlarmInfo) THEN
		fUIInRtStatHide(ADR(tyCommon.tyInfo.tyLyr.uiRtStat));
		tyCommon.tyInfo.tyStringInfo.sValue		:= '';
		tyCommon.tyInfo.tyHotspotClose.bRtCompl	:= FALSE;

	ELSIF tyCommon.tyInfo.tyHotspotClose.bRtCompl = TRUE THEN
		tyCommon.tyInfo.tyHotspotClose.bRtCompl	:= FALSE;
		fUIInRtStatHide(ADR(tyCommon.tyInfo.tyLyr.uiRtStat));

	ELSIF p_bAlarmInfo THEN
		tyCommon.tyInfo.tyStringInfo.sValue	:= p_sAlarmInfoMsg;

	END_IF

END_ACTION
```

#### Act_OptC0010RcyMsg.st
```iecst
ACTION Act_OptC0010RcyMsg:

	IF tyC0010RcyMsg.tyRcyMsg.tyHotspotClose.bRtCompl THEN
		fUIInRtStatHide(ADR(tyC0010RcyMsg.tyRcyMsg.tyLyr.uiRtStat));
		tyC0010RecoverMsg.tyHotspotClose.bRtCompl 	:= FALSE;
	END_IF

END_ACTION
```
